LIN {X 0,Y 201.195,Z 1275.243,A -85,B 0,C 180,E1 26164.19,E2 26164.19} C_VEL
LIN {X 0,Y 195.017,Z 1283.497,A -85,B 0,C 180,E1 26183.301,E2 26183.301} C_VEL
LIN {X 0,Y 194.999,Z 1283.507,A -85,B 0,C 180,E1 26196.699,E2 26196.699} C_VEL
LIN {X 0,Y 201.236,Z 1275.253,A -85,B 0,C 180,E1 26215.835,E2 26215.835} C_VEL
LIN {X 0,Y 226.879,Z 1253.045,A -85,B 0,C 180,E1 26235.936,E2 26235.936} C_VEL
LIN {X 0,Y 270.809,Z 1215.708,A -85,B 0,C 180,E1 26251.087,E2 26251.087} C_VEL
LIN {X 0,Y 321.141,Z 1165.252,A -85,B 0,C 180,E1 26260.774,E2 26260.774} C_VEL
LIN {X 0,Y 367.903,Z 1104.901,A -85,B 0,C 180,E1 26266.675,E2 26266.675} C_VEL
LIN {X 0,Y 370.039,Z 1092.442,A -85,B 0,C 180,E1 26272.536,E2 26272.536} C_VEL
LIN {X 0,Y 370.708,Z 1086.535,A -85,B 0,C 180,E1 26278.866,E2 26278.866} C_VEL
LIN {X 0,Y 369.636,Z 1091.478,A -85,B 0,C 180,E1 26286.971,E2 26286.971} C_VEL
LIN {X 0,Y 367.658,Z 1103.886,A -85,B 0,C 180,E1 26293.55,E2 26293.55} C_VEL
LIN {X 0,Y 320.637,Z 1164.15,A -85,B 0,C 180,E1 26299.642,E2 26299.642} C_VEL
LIN {X 0,Y 271.724,Z 1212.598,A -85,B 0,C 180,E1 26309.058,E2 26309.058} C_VEL
LIN {X 0,Y 254.088,Z 1227.944,A -85,B 0,C 180,E1 26313.968,E2 26313.968} C_VEL
LIN {X 0,Y 230.122,Z 1243.335,A -85,B 0,C 180,E1 26319.017,E2 26319.017} C_VEL
LIN {X 0,Y 198.588,Z 1267.683,A -85,B 0,C 180,E1 26338.072,E2 26338.072} C_VEL
LIN {X 0,Y 187.588,Z 1278.356,A -85,B 0,C 180,E1 26358.34,E2 26358.34} C_VEL
LIN {X 0,Y 187.248,Z 1279.786,A -85,B 0,C 180,E1 26372.321,E2 26372.321} C_VEL
LIN {X 0,Y 191.78,Z 1273.585,A -85,B 0,C 180,E1 26393.132,E2 26393.132} C_VEL
LIN {X 0,Y 216.378,Z 1253.744,A -85,B 0,C 180,E1 26414.497,E2 26414.497} C_VEL
LIN {X 0,Y 259.404,Z 1219.732,A -85,B 0,C 180,E1 26430.302,E2 26430.302} C_VEL
LIN {X 0,Y 309.886,Z 1172.58,A -85,B 0,C 180,E1 26440.494,E2 26440.494} C_VEL
LIN {X 0,Y 358.072,Z 1114.769,A -85,B 0,C 180,E1 26446.759,E2 26446.759} C_VEL
LIN {X 0,Y 363.326,Z 1107.025,A -85,B 0,C 180,E1 26447.549,E2 26447.549} C_VEL
LIN {X 0,Y 365.187,Z 1096.26,A -85,B 0,C 180,E1 26454,E2 26454} C_VEL
LIN {X 0,Y 366.009,Z 1093.019,A -85,B 0,C 180,E1 26461.149,E2 26461.149} C_VEL
LIN {X 0,Y 364.774,Z 1102.007,A -85,B 0,C 180,E1 26469.54,E2 26469.54} C_VEL
LIN {X 0,Y 362.75,Z 1109.497,A -85,B 0,C 180,E1 26472.412,E2 26472.412} C_VEL
LIN {X 0,Y 315.401,Z 1168.445,A -85,B 0,C 180,E1 26478.275,E2 26478.275} C_VEL
LIN {X 0,Y 264.142,Z 1217.988,A -85,B 0,C 180,E1 26488.027,E2 26488.027} C_VEL
LIN {X 0,Y 219.314,Z 1254.431,A -85,B 0,C 180,E1 26503.442,E2 26503.442} C_VEL
LIN {X 0,Y 192.773,Z 1276.213,A -85,B 0,C 180,E1 26524.651,E2 26524.651} C_VEL
LIN {X 0,Y 187.008,Z 1283.409,A -85,B 0,C 180,E1 26543.013,E2 26543.013} C_VEL
LIN {X 0,Y 186.992,Z 1283.419,A -85,B 0,C 180,E1 26556.987,E2 26556.987} C_VEL
LIN {X 0,Y 194.576,Z 1274.473,A -85,B 0,C 180,E1 26577.881,E2 26577.881} C_VEL
LIN {X 0,Y 223.086,Z 1251.404,A -85,B 0,C 180,E1 26598.398,E2 26598.398} C_VEL
LIN {X 0,Y 270.344,Z 1212.537,A -85,B 0,C 180,E1 26613.469,E2 26613.469} C_VEL
LIN {X 0,Y 321.331,Z 1162.031,A -85,B 0,C 180,E1 26622.583,E2 26622.583} C_VEL
LIN {X 0,Y 364.275,Z 1106.957,A -85,B 0,C 180,E1 26628.053,E2 26628.053} C_VEL
LIN {X 0,Y 365.739,Z 1094.84,A -85,B 0,C 180,E1 26636.472,E2 26636.472} C_VEL
LIN {X 0,Y 365.521,Z 1094.699,A -85,B 0,C 180,E1 26643.608,E2 26643.608} C_VEL
LIN {X 0,Y 363.417,Z 1106.744,A -85,B 0,C 180,E1 26652.086,E2 26652.086} C_VEL
LIN {X 0,Y 354.781,Z 1119.511,A -85,B 0,C 180,E1 26653.483,E2 26653.483} C_VEL
LIN {X 0,Y 305.533,Z 1177.31,A -85,B 0,C 180,E1 26660.141,E2 26660.141} C_VEL
LIN {X 0,Y 255.501,Z 1223.045,A -85,B 0,C 180,E1 26670.61,E2 26670.61} C_VEL
LIN {X 0,Y 230.122,Z 1243.335,A -85,B 0,C 180,E1 26679.017,E2 26679.017} C_VEL
LIN {X 0,Y 207.484,Z 1256.044,A -85,B 0,C 180,E1 26685.371,E2 26685.371} C_VEL
LIN {X 0,Y 183.024,Z 1274.859,A -85,B 0,C 180,E1 26708.108,E2 26708.108} C_VEL
LIN {X 0,Y 179.002,Z 1279.886,A -85,B 0,C 180,E1 26727.572,E2 26727.572} C_VEL
LIN {X 0,Y 180.111,Z 1277.868,A -85,B 0,C 180,E1 26744.074,E2 26744.074} C_VEL
LIN {X 0,Y 194.472,Z 1265.479,A -85,B 0,C 180,E1 26765.794,E2 26765.794} C_VEL
LIN {X 0,Y 231.406,Z 1238.37,A -85,B 0,C 180,E1 26785.005,E2 26785.005} C_VEL
LIN {X 0,Y 282.219,Z 1196.766,A -85,B 0,C 180,E1 26797.777,E2 26797.777} C_VEL
LIN {X 0,Y 334.047,Z 1143.181,A -85,B 0,C 180,E1 26805.559,E2 26805.559} C_VEL
LIN {X 0,Y 358.451,Z 1111.801,A -85,B 0,C 180,E1 26808.363,E2 26808.363} C_VEL
LIN {X 0,Y 360.648,Z 1100.805,A -85,B 0,C 180,E1 26816.343,E2 26816.343} C_VEL
LIN {X 0,Y 361.231,Z 1099.493,A -85,B 0,C 180,E1 26821.164,E2 26821.164} C_VEL
LIN {X 0,Y 359.753,Z 1108.809,A -85,B 0,C 180,E1 26829.674,E2 26829.674} C_VEL
LIN {X 0,Y 357.604,Z 1114.227,A -85,B 0,C 180,E1 26831.491,E2 26831.491} C_VEL
LIN {X 0,Y 309.713,Z 1171.72,A -85,B 0,C 180,E1 26837.286,E2 26837.286} C_VEL
LIN {X 0,Y 257.526,Z 1220.154,A -85,B 0,C 180,E1 26847.039,E2 26847.039} C_VEL
LIN {X 0,Y 211.366,Z 1255.921,A -85,B 0,C 180,E1 26862.896,E2 26862.896} C_VEL
LIN {X 0,Y 185.522,Z 1275.938,A -85,B 0,C 180,E1 26883.282,E2 26883.282} C_VEL
LIN {X 0,Y 179.001,Z 1283.32,A -85,B 0,C 180,E1 26902.699,E2 26902.699} C_VEL
LIN {X 0,Y 178.986,Z 1283.331,A -85,B 0,C 180,E1 26917.301,E2 26917.301} C_VEL
LIN {X 0,Y 187.317,Z 1274.383,A -85,B 0,C 180,E1 26939.062,E2 26939.062} C_VEL
LIN {X 0,Y 219.732,Z 1249.764,A -85,B 0,C 180,E1 26960.936,E2 26960.936} C_VEL
LIN {X 0,Y 268.261,Z 1211.154,A -85,B 0,C 180,E1 26975.394,E2 26975.394} C_VEL
LIN {X 0,Y 320.449,Z 1160.299,A -85,B 0,C 180,E1 26984.216,E2 26984.216} C_VEL
LIN {X 0,Y 359.366,Z 1111.989,A -85,B 0,C 180,E1 26988.782,E2 26988.782} C_VEL
LIN {X 0,Y 360.904,Z 1101.309,A -85,B 0,C 180,E1 26996.424,E2 26996.424} C_VEL
LIN {X 0,Y 361.206,Z 1099.765,A -85,B 0,C 180,E1 27001.242,E2 27001.242} C_VEL
LIN {X 0,Y 359.072,Z 1109.384,A -85,B 0,C 180,E1 27010.124,E2 27010.124} C_VEL
LIN {X 0,Y 356.374,Z 1114.981,A -85,B 0,C 180,E1 27011.826,E2 27011.826} C_VEL
LIN {X 0,Y 306.687,Z 1173.441,A -85,B 0,C 180,E1 27018.074,E2 27018.074} C_VEL
LIN {X 0,Y 254.942,Z 1220.25,A -85,B 0,C 180,E1 27028.066,E2 27028.066} C_VEL
LIN {X 0,Y 209.353,Z 1254.643,A -85,B 0,C 180,E1 27044.325,E2 27044.325} C_VEL
LIN {X 0,Y 207.484,Z 1256.044,A -85,B 0,C 180,E1 27045.371,E2 27045.371} C_VEL
LIN {X 0,Y 187.092,Z 1266.177,A -85,B 0,C 180,E1 27053.33,E2 27053.33} C_VEL
LIN {X 0,Y 171.751,Z 1278.533,A -85,B 0,C 180,E1 27077.247,E2 27077.247} C_VEL
LIN {X 0,Y 171.202,Z 1279.961,A -85,B 0,C 180,E1 27092.539,E2 27092.539} C_VEL
LIN {X 0,Y 175.429,Z 1274.881,A -85,B 0,C 180,E1 27112.893,E2 27112.893} C_VEL
LIN {X 0,Y 200.894,Z 1256.581,A -85,B 0,C 180,E1 27135.82,E2 27135.82} C_VEL
LIN {X 0,Y 247.578,Z 1223.011,A -85,B 0,C 180,E1 27152.648,E2 27152.648} C_VEL
LIN {X 0,Y 301.387,Z 1176.096,A -85,B 0,C 180,E1 27162.951,E2 27162.951} C_VEL
LIN {X 0,Y 352.482,Z 1117.88,A -85,B 0,C 180,E1 27169.115,E2 27169.115} C_VEL
LIN {X 0,Y 355.572,Z 1108.315,A -85,B 0,C 180,E1 27175.006,E2 27175.006} C_VEL
LIN {X 0,Y 356.408,Z 1105.935,A -85,B 0,C 180,E1 27181.18,E2 27181.18} C_VEL
LIN {X 0,Y 354.546,Z 1115.239,A -85,B 0,C 180,E1 27189.682,E2 27189.682} C_VEL
LIN {X 0,Y 350.481,Z 1121.555,A -85,B 0,C 180,E1 27190.725,E2 27190.725} C_VEL
LIN {X 0,Y 300.864,Z 1178.068,A -85,B 0,C 180,E1 27196.721,E2 27196.721} C_VEL
LIN {X 0,Y 246.815,Z 1225.533,A -85,B 0,C 180,E1 27207.008,E2 27207.008} C_VEL
LIN {X 0,Y 200.187,Z 1259.672,A -85,B 0,C 180,E1 27223.972,E2 27223.972} C_VEL
LIN {X 0,Y 175.136,Z 1278.434,A -85,B 0,C 180,E1 27247.066,E2 27247.066} C_VEL
LIN {X 0,Y 170.978,Z 1283.704,A -85,B 0,C 180,E1 27267.458,E2 27267.458} C_VEL
LIN {X 0,Y 171.647,Z 1282.189,A -85,B 0,C 180,E1 27282.76,E2 27282.76} C_VEL
LIN {X 0,Y 185.284,Z 1270.435,A -85,B 0,C 180,E1 27305.582,E2 27305.582} C_VEL
LIN {X 0,Y 223.656,Z 1243.055,A -85,B 0,C 180,E1 27326.162,E2 27326.162} C_VEL
LIN {X 0,Y 275.987,Z 1201.491,A -85,B 0,C 180,E1 27339.198,E2 27339.198} C_VEL
LIN {X 0,Y 328.939,Z 1148.262,A -85,B 0,C 180,E1 27346.968,E2 27346.968} C_VEL
LIN {X 0,Y 354.471,Z 1116.219,A -85,B 0,C 180,E1 27349.881,E2 27349.881} C_VEL
LIN {X 0,Y 356.56,Z 1106.115,A -85,B 0,C 180,E1 27358.821,E2 27358.821} C_VEL
LIN {X 0,Y 354.841,Z 1111.535,A -85,B 0,C 180,E1 27367.41,E2 27367.41} C_VEL
LIN {X 0,Y 352.623,Z 1117.947,A -85,B 0,C 180,E1 27370.75,E2 27370.75} C_VEL
LIN {X 0,Y 301.319,Z 1176.4,A -85,B 0,C 180,E1 27377.008,E2 27377.008} C_VEL
LIN {X 0,Y 247.419,Z 1223.224,A -85,B 0,C 180,E1 27387.282,E2 27387.282} C_VEL
LIN {X 0,Y 200.777,Z 1256.725,A -85,B 0,C 180,E1 27404.146,E2 27404.146} C_VEL
LIN {X 0,Y 187.092,Z 1266.177,A -85,B 0,C 180,E1 27413.33,E2 27413.33} C_VEL
LIN {X 0,Y 169.798,Z 1273.66,A -85,B 0,C 180,E1 27423.03,E2 27423.03} C_VEL
LIN {X 0,Y 163.094,Z 1279.631,A -85,B 0,C 180,E1 27441.983,E2 27441.983} C_VEL
LIN {X 0,Y 163.159,Z 1279.601,A -85,B 0,C 180,E1 27458.015,E2 27458.015} C_VEL
LIN {X 0,Y 173.522,Z 1270.917,A -85,B 0,C 180,E1 27481.627,E2 27481.627} C_VEL
LIN {X 0,Y 210.173,Z 1246.793,A -85,B 0,C 180,E1 27504.269,E2 27504.269} C_VEL
LIN {X 0,Y 262.077,Z 1208.946,A -85,B 0,C 180,E1 27518.303,E2 27518.303} C_VEL
LIN {X 0,Y 316.745,Z 1158.307,A -85,B 0,C 180,E1 27526.782,E2 27526.782} C_VEL
LIN {X 0,Y 348.764,Z 1120.766,A -85,B 0,C 180,E1 27530.367,E2 27530.367} C_VEL
LIN {X 0,Y 351.543,Z 1112.083,A -85,B 0,C 180,E1 27538.724,E2 27538.724} C_VEL
LIN {X 0,Y 350.398,Z 1116.362,A -85,B 0,C 180,E1 27546.173,E2 27546.173} C_VEL
LIN {X 0,Y 348.485,Z 1122.201,A -85,B 0,C 180,E1 27549.453,E2 27549.453} C_VEL
LIN {X 0,Y 296.939,Z 1179.584,A -85,B 0,C 180,E1 27555.422,E2 27555.422} C_VEL
LIN {X 0,Y 241.164,Z 1226.947,A -85,B 0,C 180,E1 27565.712,E2 27565.712} C_VEL
LIN {X 0,Y 194.488,Z 1259.579,A -85,B 0,C 180,E1 27582.202,E2 27582.202} C_VEL
LIN {X 0,Y 167.582,Z 1278.344,A -85,B 0,C 180,E1 27605.969,E2 27605.969} C_VEL
LIN {X 0,Y 162.958,Z 1283.617,A -85,B 0,C 180,E1 27627.333,E2 27627.333} C_VEL
LIN {X 0,Y 163.819,Z 1282.005,A -85,B 0,C 180,E1 27643.871,E2 27643.871} C_VEL
LIN {X 0,Y 180.769,Z 1268.817,A -85,B 0,C 180,E1 27668.991,E2 27668.991} C_VEL
LIN {X 0,Y 221.546,Z 1241.207,A -85,B 0,C 180,E1 27688.832,E2 27688.832} C_VEL
LIN {X 0,Y 275.798,Z 1199.137,A -85,B 0,C 180,E1 27701.284,E2 27701.284} C_VEL
LIN {X 0,Y 329.387,Z 1145.675,A -85,B 0,C 180,E1 27708.631,E2 27708.631} C_VEL
LIN {X 0,Y 349.546,Z 1120.838,A -85,B 0,C 180,E1 27710.854,E2 27710.854} C_VEL
LIN {X 0,Y 351.639,Z 1112.474,A -85,B 0,C 180,E1 27718.804,E2 27718.804} C_VEL
LIN {X 0,Y 350.023,Z 1116.409,A -85,B 0,C 180,E1 27726.261,E2 27726.261} C_VEL
LIN {X 0,Y 347.621,Z 1122.721,A -85,B 0,C 180,E1 27729.781,E2 27729.781} C_VEL
LIN {X 0,Y 295.744,Z 1179.677,A -85,B 0,C 180,E1 27735.956,E2 27735.956} C_VEL
LIN {X 0,Y 241.553,Z 1224.963,A -85,B 0,C 180,E1 27746.058,E2 27746.058} C_VEL
LIN {X 0,Y 193.133,Z 1258.137,A -85,B 0,C 180,E1 27763.42,E2 27763.42} C_VEL
LIN {X 0,Y 169.798,Z 1273.66,A -85,B 0,C 180,E1 27783.03,E2 27783.03} C_VEL
LIN {X 0,Y 156.267,Z 1278.321,A -85,B 0,C 180,E1 27794.526,E2 27794.526} C_VEL
LIN {X 0,Y 155.168,Z 1280.137,A -85,B 0,C 180,E1 27812.801,E2 27812.801} C_VEL
LIN {X 0,Y 161.274,Z 1274.488,A -85,B 0,C 180,E1 27836.473,E2 27836.473} C_VEL
LIN {X 0,Y 194.237,Z 1253.968,A -85,B 0,C 180,E1 27861.528,E2 27861.528} C_VEL
LIN {X 0,Y 244.846,Z 1219.958,A -85,B 0,C 180,E1 27877.122,E2 27877.122} C_VEL
LIN {X 0,Y 300.305,Z 1173.094,A -85,B 0,C 180,E1 27886.44,E2 27886.44} C_VEL
LIN {X 0,Y 343.984,Z 1125.372,A -85,B 0,C 180,E1 27891.399,E2 27891.399} C_VEL
LIN {X 0,Y 346.418,Z 1118.322,A -85,B 0,C 180,E1 27898.705,E2 27898.705} C_VEL
LIN {X 0,Y 345.169,Z 1122.764,A -85,B 0,C 180,E1 27906.267,E2 27906.267} C_VEL
LIN {X 0,Y 343.768,Z 1126.608,A -85,B 0,C 180,E1 27908.435,E2 27908.435} C_VEL
LIN {X 0,Y 291.229,Z 1182.986,A -85,B 0,C 180,E1 27914.361,E2 27914.361} C_VEL
LIN {X 0,Y 235.946,Z 1228.133,A -85,B 0,C 180,E1 27924.283,E2 27924.283} C_VEL
LIN {X 0,Y 186.895,Z 1260.839,A -85,B 0,C 180,E1 27941.359,E2 27941.359} C_VEL
LIN {X 0,Y 160.09,Z 1278.253,A -85,B 0,C 180,E1 27964.768,E2 27964.768} C_VEL
LIN {X 0,Y 154.936,Z 1283.529,A -85,B 0,C 180,E1 27987.195,E2 27987.195} C_VEL
LIN {X 0,Y 155.862,Z 1282.011,A -85,B 0,C 180,E1 28004.078,E2 28004.078} C_VEL
LIN {X 0,Y 172.151,Z 1270.141,A -85,B 0,C 180,E1 28028.962,E2 28028.962} C_VEL
LIN {X 0,Y 214.695,Z 1242.871,A -85,B 0,C 180,E1 28049.916,E2 28049.916} C_VEL
LIN {X 0,Y 270.961,Z 1200.936,A -85,B 0,C 180,E1 28062.579,E2 28062.579} C_VEL
LIN {X 0,Y 326.907,Z 1146.64,A -85,B 0,C 180,E1 28069.95,E2 28069.95} C_VEL
LIN {X 0,Y 344.662,Z 1125.488,A -85,B 0,C 180,E1 28071.896,E2 28071.896} C_VEL
LIN {X 0,Y 346.513,Z 1118.711,A -85,B 0,C 180,E1 28078.786,E2 28078.786} C_VEL
LIN {X 0,Y 344.788,Z 1122.817,A -85,B 0,C 180,E1 28086.356,E2 28086.356} C_VEL
LIN {X 0,Y 342.867,Z 1127.123,A -85,B 0,C 180,E1 28088.759,E2 28088.759} C_VEL
LIN {X 0,Y 289.1,Z 1183.852,A -85,B 0,C 180,E1 28095.015,E2 28095.015} C_VEL
LIN {X 0,Y 232.169,Z 1229.12,A -85,B 0,C 180,E1 28105.638,E2 28105.638} C_VEL
LIN {X 0,Y 183.612,Z 1260.51,A -85,B 0,C 180,E1 28123.722,E2 28123.722} C_VEL
LIN {X 0,Y 158.982,Z 1276.302,A -85,B 0,C 180,E1 28147.57,E2 28147.57} C_VEL
LIN {X 0,Y 156.267,Z 1278.321,A -85,B 0,C 180,E1 28154.526,E2 28154.526} C_VEL
LIN {X 0,Y 146.914,Z 1280.235,A -85,B 0,C 180,E1 28167.516,E2 28167.516} C_VEL
LIN {X 0,Y 148.18,Z 1278.77,A -85,B 0,C 180,E1 28184.825,E2 28184.825} C_VEL
LIN {X 0,Y 165.314,Z 1267.75,A -85,B 0,C 180,E1 28209.953,E2 28209.953} C_VEL
LIN {X 0,Y 208.556,Z 1242.191,A -85,B 0,C 180,E1 28230.761,E2 28230.761} C_VEL
LIN {X 0,Y 265.721,Z 1201.741,A -85,B 0,C 180,E1 28243.402,E2 28243.402} C_VEL
LIN {X 0,Y 321.32,Z 1150.153,A -85,B 0,C 180,E1 28250.545,E2 28250.545} C_VEL
LIN {X 0,Y 339.042,Z 1129.89,A -85,B 0,C 180,E1 28252.482,E2 28252.482} C_VEL
LIN {X 0,Y 341.255,Z 1124.682,A -85,B 0,C 180,E1 28260.805,E2 28260.805} C_VEL
LIN {X 0,Y 338.694,Z 1131.184,A -85,B 0,C 180,E1 28267.412,E2 28267.412} C_VEL
LIN {X 0,Y 284.233,Z 1187.296,A -85,B 0,C 180,E1 28273.42,E2 28273.42} C_VEL
LIN {X 0,Y 227.106,Z 1231.739,A -85,B 0,C 180,E1 28283.658,E2 28283.658} C_VEL
LIN {X 0,Y 177.311,Z 1263.096,A -85,B 0,C 180,E1 28301.549,E2 28301.549} C_VEL
LIN {X 0,Y 151.147,Z 1279.385,A -85,B 0,C 180,E1 28326.338,E2 28326.338} C_VEL
LIN {X 0,Y 146.914,Z 1283.441,A -85,B 0,C 180,E1 28347.041,E2 28347.041} C_VEL
LIN {X 0,Y 147.995,Z 1281.923,A -85,B 0,C 180,E1 28364.843,E2 28364.843} C_VEL
LIN {X 0,Y 168.083,Z 1268.635,A -85,B 0,C 180,E1 28392.585,E2 28392.585} C_VEL
LIN {X 0,Y 213.321,Z 1241.025,A -85,B 0,C 180,E1 28412.703,E2 28412.703} C_VEL
LIN {X 0,Y 271.233,Z 1198.685,A -85,B 0,C 180,E1 28424.686,E2 28424.686} C_VEL
LIN {X 0,Y 327.503,Z 1144.437,A -85,B 0,C 180,E1 28431.575,E2 28431.575} C_VEL
LIN {X 0,Y 339.627,Z 1130.078,A -85,B 0,C 180,E1 28432.994,E2 28432.994} C_VEL
LIN {X 0,Y 341.24,Z 1124.941,A -85,B 0,C 180,E1 28440.615,E2 28440.615} C_VEL
LIN {X 0,Y 338.878,Z 1130.436,A -85,B 0,C 180,E1 28447.529,E2 28447.529} C_VEL
LIN {X 0,Y 284.419,Z 1186.22,A -85,B 0,C 180,E1 28453.76,E2 28453.76} C_VEL
LIN {X 0,Y 226.913,Z 1230.379,A -85,B 0,C 180,E1 28464.17,E2 28464.17} C_VEL
LIN {X 0,Y 175.98,Z 1261.736,A -85,B 0,C 180,E1 28482.904,E2 28482.904} C_VEL
LIN {X 0,Y 150.076,Z 1277.237,A -85,B 0,C 180,E1 28509.288,E2 28509.288} C_VEL
LIN {X 0,Y 146.914,Z 1280.235,A -85,B 0,C 180,E1 28527.516,E2 28527.516} C_VEL
LIN {X 0,Y 139.41,Z 1279.532,A -85,B 0,C 180,E1 28541.496,E2 28541.496} C_VEL
LIN {X 0,Y 155.826,Z 1269.649,A -85,B 0,C 180,E1 28569.242,E2 28569.242} C_VEL
LIN {X 0,Y 199.179,Z 1245.552,A -85,B 0,C 180,E1 28591.117,E2 28591.117} C_VEL
LIN {X 0,Y 257.986,Z 1206.184,A -85,B 0,C 180,E1 28604.278,E2 28604.278} C_VEL
LIN {X 0,Y 316.518,Z 1154.072,A -85,B 0,C 180,E1 28611.654,E2 28611.654} C_VEL
LIN {X 0,Y 334.007,Z 1134.744,A -85,B 0,C 180,E1 28613.438,E2 28613.438} C_VEL
LIN {X 0,Y 335.952,Z 1130.602,A -85,B 0,C 180,E1 28618.664,E2 28618.664} C_VEL
LIN {X 0,Y 334.42,Z 1134.828,A -85,B 0,C 180,E1 28626.142,E2 28626.142} C_VEL
LIN {X 0,Y 277.384,Z 1191.533,A -85,B 0,C 180,E1 28632.432,E2 28632.432} C_VEL
LIN {X 0,Y 218.28,Z 1235.316,A -85,B 0,C 180,E1 28642.991,E2 28642.991} C_VEL
LIN {X 0,Y 169.75,Z 1264.166,A -85,B 0,C 180,E1 28660.59,E2 28660.59} C_VEL
LIN {X 0,Y 142.215,Z 1280.182,A -85,B 0,C 180,E1 28688.085,E2 28688.085} C_VEL
LIN {X 0,Y 138.905,Z 1283.353,A -85,B 0,C 180,E1 28706.87,E2 28706.87} C_VEL
LIN {X 0,Y 140.139,Z 1281.834,A -85,B 0,C 180,E1 28725.696,E2 28725.696} C_VEL
LIN {X 0,Y 158.595,Z 1270.499,A -85,B 0,C 180,E1 28752.017,E2 28752.017} C_VEL
LIN {X 0,Y 205.375,Z 1243.558,A -85,B 0,C 180,E1 28773.563,E2 28773.563} C_VEL
LIN {X 0,Y 264.133,Z 1202.601,A -85,B 0,C 180,E1 28785.67,E2 28785.67} C_VEL
LIN {X 0,Y 321.204,Z 1149.944,A -85,B 0,C 180,E1 28792.521,E2 28792.521} C_VEL
LIN {X 0,Y 334.47,Z 1135.059,A -85,B 0,C 180,E1 28793.858,E2 28793.858} C_VEL
LIN {X 0,Y 335.817,Z 1131.076,A -85,B 0,C 180,E1 28801.336,E2 28801.336} C_VEL
LIN {X 0,Y 332.534,Z 1136.844,A -85,B 0,C 180,E1 28806.743,E2 28806.743} C_VEL
LIN {X 0,Y 276.142,Z 1191.82,A -85,B 0,C 180,E1 28813,E2 28813} C_VEL
LIN {X 0,Y 218.878,Z 1233.575,A -85,B 0,C 180,E1 28823.358,E2 28823.358} C_VEL
LIN {X 0,Y 168.05,Z 1263.152,A -85,B 0,C 180,E1 28842.206,E2 28842.206} C_VEL
LIN {X 0,Y 142.461,Z 1277.326,A -85,B 0,C 180,E1 28868.125,E2 28868.125} C_VEL
LIN {X 0,Y 138.887,Z 1280.323,A -85,B 0,C 180,E1 28887.418,E2 28887.418} C_VEL
LIN {X 0,Y 139.41,Z 1279.532,A -85,B 0,C 180,E1 28901.496,E2 28901.496} C_VEL
LIN {X 0,Y 136.452,Z 1276.545,A -85,B 0,C 180,E1 28916.168,E2 28916.168} C_VEL
LIN {X 0,Y 171.443,Z 1258.694,A -85,B 0,C 180,E1 28944.33,E2 28944.33} C_VEL
LIN {X 0,Y 227.496,Z 1226.156,A -85,B 0,C 180,E1 28961.07,E2 28961.07} C_VEL
LIN {X 0,Y 287.562,Z 1180.546,A -85,B 0,C 180,E1 28970.248,E2 28970.248} C_VEL
LIN {X 0,Y 329.132,Z 1139.395,A -85,B 0,C 180,E1 28974.666,E2 28974.666} C_VEL
LIN {X 0,Y 330.526,Z 1136.788,A -85,B 0,C 180,E1 28981.272,E2 28981.272} C_VEL
LIN {X 0,Y 328.525,Z 1140.754,A -85,B 0,C 180,E1 28985.322,E2 28985.322} C_VEL
LIN {X 0,Y 270.712,Z 1195.661,A -85,B 0,C 180,E1 28991.375,E2 28991.375} C_VEL
LIN {X 0,Y 209.11,Z 1238.993,A -85,B 0,C 180,E1 29002.38,E2 29002.38} C_VEL
LIN {X 0,Y 159.07,Z 1266.951,A -85,B 0,C 180,E1 29021.377,E2 29021.377} C_VEL
LIN {X 0,Y 134.657,Z 1280.092,A -85,B 0,C 180,E1 29046.785,E2 29046.785} C_VEL
LIN {X 0,Y 130.881,Z 1283.265,A -85,B 0,C 180,E1 29066.678,E2 29066.678} C_VEL
LIN {X 0,Y 132.327,Z 1281.745,A -85,B 0,C 180,E1 29086.649,E2 29086.649} C_VEL
LIN {X 0,Y 152.475,Z 1270.408,A -85,B 0,C 180,E1 29114.125,E2 29114.125} C_VEL
LIN {X 0,Y 201.405,Z 1243.688,A -85,B 0,C 180,E1 29135.603,E2 29135.603} C_VEL
LIN {X 0,Y 262.201,Z 1202.513,A -85,B 0,C 180,E1 29147.429,E2 29147.429} C_VEL
LIN {X 0,Y 320.231,Z 1149.856,A -85,B 0,C 180,E1 29153.992,E2 29153.992} C_VEL
LIN {X 0,Y 329.451,Z 1139.81,A -85,B 0,C 180,E1 29155.011,E2 29155.011} C_VEL
LIN {X 0,Y 330.414,Z 1137.075,A -85,B 0,C 180,E1 29161.358,E2 29161.358} C_VEL
LIN {X 0,Y 327.668,Z 1141.474,A -85,B 0,C 180,E1 29165.688,E2 29165.688} C_VEL
LIN {X 0,Y 269.343,Z 1195.997,A -85,B 0,C 180,E1 29171.959,E2 29171.959} C_VEL
LIN {X 0,Y 209.726,Z 1237.359,A -85,B 0,C 180,E1 29182.787,E2 29182.787} C_VEL
LIN {X 0,Y 160.681,Z 1264.266,A -85,B 0,C 180,E1 29201.115,E2 29201.115} C_VEL
LIN {X 0,Y 134.903,Z 1277.416,A -85,B 0,C 180,E1 29226.83,E2 29226.83} C_VEL
LIN {X 0,Y 130.914,Z 1280.412,A -85,B 0,C 180,E1 29246.68,E2 29246.68} C_VEL
LIN {X 0,Y 132.527,Z 1278.948,A -85,B 0,C 180,E1 29266.624,E2 29266.624} C_VEL
LIN {X 0,Y 136.452,Z 1276.545,A -85,B 0,C 180,E1 29276.168,E2 29276.168} C_VEL
LIN {X 0,Y 140.06,Z 1271.301,A -85,B 0,C 180,E1 29290.712,E2 29290.712} C_VEL
LIN {X 0,Y 186.683,Z 1248.373,A -85,B 0,C 180,E1 29314.029,E2 29314.029} C_VEL
LIN {X 0,Y 247.881,Z 1210.661,A -85,B 0,C 180,E1 29327.007,E2 29327.007} C_VEL
LIN {X 0,Y 308.358,Z 1160.282,A -85,B 0,C 180,E1 29334.086,E2 29334.086} C_VEL
LIN {X 0,Y 323.904,Z 1144.401,A -85,B 0,C 180,E1 29335.583,E2 29335.583} C_VEL
LIN {X 0,Y 325.054,Z 1142.71,A -85,B 0,C 180,E1 29341.294,E2 29341.294} C_VEL
LIN {X 0,Y 322.953,Z 1145.849,A -85,B 0,C 180,E1 29344.261,E2 29344.261} C_VEL
LIN {X 0,Y 263.951,Z 1199.577,A -85,B 0,C 180,E1 29350.287,E2 29350.287} C_VEL
LIN {X 0,Y 202.984,Z 1240.653,A -85,B 0,C 180,E1 29360.948,E2 29360.948} C_VEL
LIN {X 0,Y 150.53,Z 1268.309,A -85,B 0,C 180,E1 29380.922,E2 29380.922} C_VEL
LIN {X 0,Y 127.143,Z 1280.002,A -85,B 0,C 180,E1 29405.324,E2 29405.324} C_VEL
LIN {X 0,Y 122.857,Z 1283.177,A -85,B 0,C 180,E1 29426.461,E2 29426.461} C_VEL
LIN {X 0,Y 124.538,Z 1281.656,A -85,B 0,C 180,E1 29447.724,E2 29447.724} C_VEL
LIN {X 0,Y 146.586,Z 1270.318,A -85,B 0,C 180,E1 29476.402,E2 29476.402} C_VEL
LIN {X 0,Y 198.08,Z 1243.597,A -85,B 0,C 180,E1 29497.819,E2 29497.819} C_VEL
LIN {X 0,Y 260.501,Z 1202.423,A -85,B 0,C 180,E1 29509.233,E2 29509.233} C_VEL
LIN {X 0,Y 319.934,Z 1149.281,A -85,B 0,C 180,E1 29515.509,E2 29515.509} C_VEL
LIN {X 0,Y 324.216,Z 1144.711,A -85,B 0,C 180,E1 29516.019,E2 29516.019} C_VEL
LIN {X 0,Y 324.903,Z 1142.997,A -85,B 0,C 180,E1 29521.381,E2 29521.381} C_VEL
LIN {X 0,Y 322.828,Z 1145.866,A -85,B 0,C 180,E1 29524.596,E2 29524.596} C_VEL
LIN {X 0,Y 264.259,Z 1198.727,A -85,B 0,C 180,E1 29530.651,E2 29530.651} C_VEL
LIN {X 0,Y 203.563,Z 1239.174,A -85,B 0,C 180,E1 29541.371,E2 29541.371} C_VEL
LIN {X 0,Y 151.179,Z 1266.214,A -85,B 0,C 180,E1 29561.206,E2 29561.206} C_VEL
LIN {X 0,Y 124.682,Z 1279.065,A -85,B 0,C 180,E1 29592.297,E2 29592.297} C_VEL
LIN {X 0,Y 123.097,Z 1280.489,A -85,B 0,C 180,E1 29613.532,E2 29613.532} C_VEL
LIN {X 0,Y 133.983,Z 1274.233,A -85,B 0,C 180,E1 29644.468,E2 29644.468} C_VEL
LIN {X 0,Y 140.06,Z 1271.301,A -85,B 0,C 180,E1 29650.712,E2 29650.712} C_VEL
LIN {X 0,Y 150.441,Z 1264.214,A -85,B 0,C 180,E1 29663.852,E2 29663.852} C_VEL
LIN {X 0,Y 207.041,Z 1235.613,A -85,B 0,C 180,E1 29682.219,E2 29682.219} C_VEL
LIN {X 0,Y 269.348,Z 1193.708,A -85,B 0,C 180,E1 29691.853,E2 29691.853} C_VEL
LIN {X 0,Y 318.654,Z 1149.326,A -85,B 0,C 180,E1 29696.823,E2 29696.823} C_VEL
LIN {X 0,Y 318.824,Z 1149.441,A -85,B 0,C 180,E1 29702.859,E2 29702.859} C_VEL
LIN {X 0,Y 258.114,Z 1202.872,A -85,B 0,C 180,E1 29709.052,E2 29709.052} C_VEL
LIN {X 0,Y 195.289,Z 1243.278,A -85,B 0,C 180,E1 29719.846,E2 29719.846} C_VEL
LIN {X 0,Y 140.875,Z 1270.198,A -85,B 0,C 180,E1 29741.161,E2 29741.161} C_VEL
LIN {X 0,Y 116.789,Z 1281.552,A -85,B 0,C 180,E1 29771.056,E2 29771.056} C_VEL
LIN {X 0,Y 114.787,Z 1283.093,A -85,B 0,C 180,E1 29793.787,E2 29793.787} C_VEL
LIN {X 0,Y 124.074,Z 1277.834,A -85,B 0,C 180,E1 29823.368,E2 29823.368} C_VEL
LIN {X 0,Y 167.664,Z 1257.751,A -85,B 0,C 180,E1 29851.872,E2 29851.872} C_VEL
LIN {X 0,Y 229.532,Z 1222.906,A -85,B 0,C 180,E1 29866.885,E2 29866.885} C_VEL
LIN {X 0,Y 291.777,Z 1175.648,A -85,B 0,C 180,E1 29874.599,E2 29874.599} C_VEL
LIN {X 0,Y 318.848,Z 1149.706,A -85,B 0,C 180,E1 29877.097,E2 29877.097} C_VEL
LIN {X 0,Y 318.096,Z 1150.27,A -85,B 0,C 180,E1 29883.461,E2 29883.461} C_VEL
LIN {X 0,Y 257.568,Z 1202.777,A -85,B 0,C 180,E1 29889.522,E2 29889.522} C_VEL
LIN {X 0,Y 194.372,Z 1242.755,A -85,B 0,C 180,E1 29900.639,E2 29900.639} C_VEL
LIN {X 0,Y 141.514,Z 1268.207,A -85,B 0,C 180,E1 29921.396,E2 29921.396} C_VEL
LIN {X 0,Y 116.96,Z 1279.154,A -85,B 0,C 180,E1 29951.086,E2 29951.086} C_VEL
LIN {X 0,Y 115.068,Z 1280.577,A -85,B 0,C 180,E1 29973.779,E2 29973.779} C_VEL
LIN {X 0,Y 127.271,Z 1274.324,A -85,B 0,C 180,E1 30006.569,E2 30006.569} C_VEL
LIN {X 0,Y 150.441,Z 1264.214,A -85,B 0,C 180,E1 30023.852,E2 30023.852} C_VEL
LIN {X 0,Y 166.641,Z 1254.962,A -85,B 0,C 180,E1 30034.835,E2 30034.835} C_VEL
LIN {X 0,Y 229.885,Z 1220.605,A -85,B 0,C 180,E1 30048.708,E2 30048.708} C_VEL
LIN {X 0,Y 292.205,Z 1174.056,A -85,B 0,C 180,E1 30055.897,E2 30055.897} C_VEL
LIN {X 0,Y 313.363,Z 1154.488,A -85,B 0,C 180,E1 30057.813,E2 30057.813} C_VEL
LIN {X 0,Y 312.34,Z 1155.735,A -85,B 0,C 180,E1 30062.027,E2 30062.027} C_VEL
LIN {X 0,Y 249.881,Z 1207.946,A -85,B 0,C 180,E1 30068.067,E2 30068.067} C_VEL
LIN {X 0,Y 184.826,Z 1247.299,A -85,B 0,C 180,E1 30079.334,E2 30079.334} C_VEL
LIN {X 0,Y 131.29,Z 1271.935,A -85,B 0,C 180,E1 30101.338,E2 30101.338} C_VEL
LIN {X 0,Y 109.094,Z 1281.463,A -85,B 0,C 180,E1 30129.663,E2 30129.663} C_VEL
LIN {X 0,Y 106.782,Z 1283.005,A -85,B 0,C 180,E1 30154.072,E2 30154.072} C_VEL
LIN {X 0,Y 117.26,Z 1277.744,A -85,B 0,C 180,E1 30185.59,E2 30185.59} C_VEL
LIN {X 0,Y 163.245,Z 1257.96,A -85,B 0,C 180,E1 30214.24,E2 30214.24} C_VEL
LIN {X 0,Y 225.726,Z 1224.116,A -85,B 0,C 180,E1 30228.625,E2 30228.625} C_VEL
LIN {X 0,Y 290.126,Z 1176.42,A -85,B 0,C 180,E1 30236.139,E2 30236.139} C_VEL
LIN {X 0,Y 313.649,Z 1154.622,A -85,B 0,C 180,E1 30238.33,E2 30238.33} C_VEL
LIN {X 0,Y 312.245,Z 1155.898,A -85,B 0,C 180,E1 30242.388,E2 30242.388} C_VEL
LIN {X 0,Y 250.619,Z 1207.002,A -85,B 0,C 180,E1 30248.379,E2 30248.379} C_VEL
LIN {X 0,Y 188.455,Z 1244.543,A -85,B 0,C 180,E1 30259.037,E2 30259.037} C_VEL
LIN {X 0,Y 131.798,Z 1270.088,A -85,B 0,C 180,E1 30281.59,E2 30281.59} C_VEL
LIN {X 0,Y 109.282,Z 1279.243,A -85,B 0,C 180,E1 30309.701,E2 30309.701} C_VEL
LIN {X 0,Y 107.044,Z 1280.665,A -85,B 0,C 180,E1 30334.062,E2 30334.062} C_VEL
LIN {X 0,Y 120.723,Z 1274.415,A -85,B 0,C 180,E1 30368.911,E2 30368.911} C_VEL
LIN {X 0,Y 166.641,Z 1254.962,A -85,B 0,C 180,E1 30394.835,E2 30394.835} C_VEL
LIN {X 0,Y 186.864,Z 1243.975,A -85,B 0,C 180,E1 30403.62,E2 30403.62} C_VEL
LIN {X 0,Y 253.228,Z 1204.296,A -85,B 0,C 180,E1 30413.882,E2 30413.882} C_VEL
LIN {X 0,Y 307.875,Z 1159.554,A -85,B 0,C 180,E1 30418.895,E2 30418.895} C_VEL
LIN {X 0,Y 306.784,Z 1160.665,A -85,B 0,C 180,E1 30420.88,E2 30420.88} C_VEL
LIN {X 0,Y 244.3,Z 1210.897,A -85,B 0,C 180,E1 30426.672,E2 30426.672} C_VEL
LIN {X 0,Y 178.894,Z 1248.806,A -85,B 0,C 180,E1 30437.632,E2 30437.632} C_VEL
LIN {X 0,Y 121.64,Z 1273.435,A -85,B 0,C 180,E1 30461.578,E2 30461.578} C_VEL
LIN {X 0,Y 99.398,Z 1282.434,A -85,B 0,C 180,E1 30496.77,E2 30496.77} C_VEL
LIN {X 0,Y 99.4,Z 1282.449,A -85,B 0,C 180,E1 30523.229,E2 30523.229} C_VEL
LIN {X 0,Y 121.643,Z 1273.482,A -85,B 0,C 180,E1 30558.419,E2 30558.419} C_VEL
LIN {X 0,Y 178.921,Z 1248.894,A -85,B 0,C 180,E1 30582.366,E2 30582.366} C_VEL
LIN {X 0,Y 244.227,Z 1211.109,A -85,B 0,C 180,E1 30593.319,E2 30593.319} C_VEL
LIN {X 0,Y 306.793,Z 1160.918,A -85,B 0,C 180,E1 30599.104,E2 30599.104} C_VEL
LIN {X 0,Y 306.565,Z 1161.042,A -85,B 0,C 180,E1 30601.268,E2 30601.268} C_VEL
LIN {X 0,Y 243.812,Z 1210.891,A -85,B 0,C 180,E1 30607.138,E2 30607.138} C_VEL
LIN {X 0,Y 179.473,Z 1247.67,A -85,B 0,C 180,E1 30618.082,E2 30618.082} C_VEL
LIN {X 0,Y 122.067,Z 1271.721,A -85,B 0,C 180,E1 30641.805,E2 30641.805} C_VEL
LIN {X 0,Y 99.526,Z 1280.336,A -85,B 0,C 180,E1 30676.788,E2 30676.788} C_VEL
LIN {X 0,Y 99.593,Z 1280.31,A -85,B 0,C 180,E1 30703.204,E2 30703.204} C_VEL
LIN {X 0,Y 122.055,Z 1271.649,A -85,B 0,C 180,E1 30738.203,E2 30738.203} C_VEL
LIN {X 0,Y 176.267,Z 1249.058,A -85,B 0,C 180,E1 30761.157,E2 30761.157} C_VEL
LIN {X 0,Y 186.864,Z 1243.975,A -85,B 0,C 180,E1 30763.62,E2 30763.62} C_VEL
LIN {X 0,Y 209.945,Z 1230.845,A -85,B 0,C 180,E1 30770.439,E2 30770.439} C_VEL
LIN {X 0,Y 276.937,Z 1186.217,A -85,B 0,C 180,E1 30778.004,E2 30778.004} C_VEL
LIN {X 0,Y 300.269,Z 1166.599,A -85,B 0,C 180,E1 30779.783,E2 30779.783} C_VEL
LIN {X 0,Y 236.168,Z 1215.649,A -85,B 0,C 180,E1 30785.542,E2 30785.542} C_VEL
LIN {X 0,Y 169.824,Z 1251.883,A -85,B 0,C 180,E1 30796.615,E2 30796.615} C_VEL
LIN {X 0,Y 111.919,Z 1274.934,A -85,B 0,C 180,E1 30821.817,E2 30821.817} C_VEL
LIN {X 0,Y 91.513,Z 1282.345,A -85,B 0,C 180,E1 30855.606,E2 30855.606} C_VEL
LIN {X 0,Y 91.516,Z 1282.361,A -85,B 0,C 180,E1 30884.392,E2 30884.392} C_VEL
LIN {X 0,Y 116.254,Z 1273.391,A -85,B 0,C 180,E1 30921.508,E2 30921.508} C_VEL
LIN {X 0,Y 176.389,Z 1248.88,A -85,B 0,C 180,E1 30944.933,E2 30944.933} C_VEL
LIN {X 0,Y 244.758,Z 1210.124,A -85,B 0,C 180,E1 30955.406,E2 30955.406} C_VEL
LIN {X 0,Y 298.469,Z 1168.527,A -85,B 0,C 180,E1 30960.286,E2 30960.286} C_VEL
LIN {X 0,Y 232.707,Z 1217.642,A -85,B 0,C 180,E1 30966.368,E2 30966.368} C_VEL
LIN {X 0,Y 167.251,Z 1252.319,A -85,B 0,C 180,E1 30977.81,E2 30977.81} C_VEL
LIN {X 0,Y 112.313,Z 1273.355,A -85,B 0,C 180,E1 31002.043,E2 31002.043} C_VEL
LIN {X 0,Y 91.65,Z 1280.424,A -85,B 0,C 180,E1 31035.629,E2 31035.629} C_VEL
LIN {X 0,Y 91.717,Z 1280.399,A -85,B 0,C 180,E1 31064.361,E2 31064.361} C_VEL
LIN {X 0,Y 116.681,Z 1271.74,A -85,B 0,C 180,E1 31101.246,E2 31101.246} C_VEL
LIN {X 0,Y 173.745,Z 1249.151,A -85,B 0,C 180,E1 31123.769,E2 31123.769} C_VEL
LIN {X 0,Y 209.945,Z 1230.845,A -85,B 0,C 180,E1 31130.439,E2 31130.439} C_VEL
LIN {X 0,Y 234.416,Z 1216,A -85,B 0,C 180,E1 31135.892,E2 31135.892} C_VEL
LIN {X 0,Y 277.406,Z 1185.824,A -85,B 0,C 180,E1 31139.78,E2 31139.78} C_VEL
LIN {X 0,Y 210.029,Z 1230.654,A -85,B 0,C 180,E1 31146.522,E2 31146.522} C_VEL
LIN {X 0,Y 142.031,Z 1262.355,A -85,B 0,C 180,E1 31160.887,E2 31160.887} C_VEL
LIN {X 0,Y 94.511,Z 1278.66,A -85,B 0,C 180,E1 31190.07,E2 31190.07} C_VEL
LIN {X 0,Y 82.811,Z 1282.737,A -85,B 0,C 180,E1 31224.746,E2 31224.746} C_VEL
LIN {X 0,Y 86.55,Z 1281.211,A -85,B 0,C 180,E1 31255.979,E2 31255.979} C_VEL
LIN {X 0,Y 123.674,Z 1269.091,A -85,B 0,C 180,E1 31291.953,E2 31291.953} C_VEL
LIN {X 0,Y 188.485,Z 1242.055,A -85,B 0,C 180,E1 31310.273,E2 31310.273} C_VEL
LIN {X 0,Y 256.939,Z 1201.311,A -85,B 0,C 180,E1 31318.567,E2 31318.567} C_VEL
LIN {X 0,Y 275.821,Z 1187.263,A -85,B 0,C 180,E1 31320.297,E2 31320.297} C_VEL
LIN {X 0,Y 209.021,Z 1230.895,A -85,B 0,C 180,E1 31327.101,E2 31327.101} C_VEL
LIN {X 0,Y 142.355,Z 1261.326,A -85,B 0,C 180,E1 31341.228,E2 31341.228} C_VEL
LIN {X 0,Y 94.933,Z 1277.107,A -85,B 0,C 180,E1 31370.284,E2 31370.284} C_VEL
LIN {X 0,Y 82.837,Z 1280.939,A -85,B 0,C 180,E1 31404.748,E2 31404.748} C_VEL
LIN {X 0,Y 86.831,Z 1279.484,A -85,B 0,C 180,E1 31435.89,E2 31435.89} C_VEL
LIN {X 0,Y 127.602,Z 1266.582,A -85,B 0,C 180,E1 31473.046,E2 31473.046} C_VEL
LIN {X 0,Y 192.319,Z 1239.485,A -85,B 0,C 180,E1 31490.297,E2 31490.297} C_VEL
LIN {X 0,Y 234.416,Z 1216,A -85,B 0,C 180,E1 31495.892,E2 31495.892} C_VEL
LIN {X 0,Y 250.199,Z 1205.689,A -85,B 0,C 180,E1 31499.406,E2 31499.406} C_VEL
LIN {X 0,Y 253.061,Z 1203.699,A -85,B 0,C 180,E1 31499.875,E2 31499.875} C_VEL
LIN {X 0,Y 183.176,Z 1243.84,A -85,B 0,C 180,E1 31507.841,E2 31507.841} C_VEL
LIN {X 0,Y 117.77,Z 1269.682,A -85,B 0,C 180,E1 31525.535,E2 31525.535} C_VEL
LIN {X 0,Y 79.241,Z 1281.104,A -85,B 0,C 180,E1 31561.415,E2 31561.415} C_VEL
LIN {X 0,Y 74.733,Z 1282.654,A -85,B 0,C 180,E1 31595.823,E2 31595.823} C_VEL
LIN {X 0,Y 92.375,Z 1277.384,A -85,B 0,C 180,E1 31637.626,E2 31637.626} C_VEL
LIN {X 0,Y 153.248,Z 1256.977,A -85,B 0,C 180,E1 31666.099,E2 31666.099} C_VEL
LIN {X 0,Y 223.024,Z 1222.898,A -85,B 0,C 180,E1 31677.324,E2 31677.324} C_VEL
LIN {X 0,Y 252.896,Z 1204.006,A -85,B 0,C 180,E1 31680.322,E2 31680.322} C_VEL
LIN {X 0,Y 183.903,Z 1243.167,A -85,B 0,C 180,E1 31688.286,E2 31688.286} C_VEL
LIN {X 0,Y 118.916,Z 1268.413,A -85,B 0,C 180,E1 31705.721,E2 31705.721} C_VEL
LIN {X 0,Y 79.509,Z 1279.599,A -85,B 0,C 180,E1 31741.521,E2 31741.521} C_VEL
LIN {X 0,Y 74.996,Z 1281.017,A -85,B 0,C 180,E1 31775.804,E2 31775.804} C_VEL
LIN {X 0,Y 92.794,Z 1275.968,A -85,B 0,C 180,E1 31817.345,E2 31817.345} C_VEL
LIN {X 0,Y 153.198,Z 1256.193,A -85,B 0,C 180,E1 31845.572,E2 31845.572} C_VEL
LIN {X 0,Y 224.023,Z 1221.972,A -85,B 0,C 180,E1 31856.876,E2 31856.876} C_VEL
LIN {X 0,Y 250.199,Z 1205.689,A -85,B 0,C 180,E1 31859.406,E2 31859.406} C_VEL
LIN {X 0,Y 220.093,Z 1224.217,A -85,B 0,C 180,E1 31860.801,E2 31860.801} C_VEL
LIN {X 0,Y 148.885,Z 1257.783,A -85,B 0,C 180,E1 31871.34,E2 31871.34} C_VEL
LIN {X 0,Y 86.987,Z 1277.253,A -85,B 0,C 180,E1 31898.322,E2 31898.322} C_VEL
LIN {X 0,Y 66.776,Z 1282.561,A -85,B 0,C 180,E1 31943.479,E2 31943.479} C_VEL
LIN {X 0,Y 72.196,Z 1281.032,A -85,B 0,C 180,E1 31981.677,E2 31981.677} C_VEL
LIN {X 0,Y 120.532,Z 1267.726,A -85,B 0,C 180,E1 32020.673,E2 32020.673} C_VEL
LIN {X 0,Y 190.069,Z 1240.121,A -85,B 0,C 180,E1 32035.83,E2 32035.83} C_VEL
LIN {X 0,Y 229.737,Z 1218.787,A -85,B 0,C 180,E1 32040.309,E2 32040.309} C_VEL
LIN {X 0,Y 161.359,Z 1252.589,A -85,B 0,C 180,E1 32049.306,E2 32049.306} C_VEL
LIN {X 0,Y 97.431,Z 1273.625,A -85,B 0,C 180,E1 32071.121,E2 32071.121} C_VEL
LIN {X 0,Y 68.337,Z 1280.69,A -85,B 0,C 180,E1 32110.557,E2 32110.557} C_VEL
LIN {X 0,Y 66.996,Z 1281.105,A -85,B 0,C 180,E1 32136.499,E2 32136.499} C_VEL
LIN {X 0,Y 90.223,Z 1275.351,A -85,B 0,C 180,E1 32183.756,E2 32183.756} C_VEL
LIN {X 0,Y 151.327,Z 1256.285,A -85,B 0,C 180,E1 32208.647,E2 32208.647} C_VEL
LIN {X 0,Y 223.547,Z 1222.166,A -85,B 0,C 180,E1 32218.993,E2 32218.993} C_VEL
LIN {X 0,Y 231.383,Z 1217.687,A -85,B 0,C 180,E1 32219.759,E2 32219.759} C_VEL
LIN {X 0,Y 220.093,Z 1224.217,A -85,B 0,C 180,E1 32220.801,E2 32220.801} C_VEL
LIN {X 0,Y 202.431,Z 1233.584,A -85,B 0,C 180,E1 32219.196,E2 32219.196} C_VEL
LIN {X 0,Y 199.821,Z 1234.919,A -85,B 0,C 180,E1 32218.859,E2 32218.859} C_VEL
LIN {X 0,Y 127.125,Z 1264.228,A -85,B 0,C 180,E1 32206.445,E2 32206.445} C_VEL
LIN {X 0,Y 73.072,Z 1278.181,A -85,B 0,C 180,E1 32176.586,E2 32176.586} C_VEL
LIN {X 0,Y 58.983,Z 1281.194,A -85,B 0,C 180,E1 32137.387,E2 32137.387} C_VEL
LIN {X 0,Y 66.093,Z 1279.703,A -85,B 0,C 180,E1 32093.811,E2 32093.811} C_VEL
LIN {X 0,Y 118.362,Z 1266.938,A -85,B 0,C 180,E1 32056.066,E2 32056.066} C_VEL
LIN {X 0,Y 189.698,Z 1239.896,A -85,B 0,C 180,E1 32042.136,E2 32042.136} C_VEL
LIN {X 0,Y 204.732,Z 1232.556,A -85,B 0,C 180,E1 32039.982,E2 32039.982} C_VEL
LIN {X 0,Y 131.627,Z 1263.321,A -85,B 0,C 180,E1 32028.328,E2 32028.328} C_VEL
LIN {X 0,Y 72.725,Z 1279.309,A -85,B 0,C 180,E1 31996.874,E2 31996.874} C_VEL
LIN {X 0,Y 58.724,Z 1282.477,A -85,B 0,C 180,E1 31957.418,E2 31957.418} C_VEL
LIN {X 0,Y 65.963,Z 1280.814,A -85,B 0,C 180,E1 31913.245,E2 31913.245} C_VEL
LIN {X 0,Y 118.066,Z 1267.57,A -85,B 0,C 180,E1 31875.556,E2 31875.556} C_VEL
LIN {X 0,Y 189.645,Z 1239.906,A -85,B 0,C 180,E1 31861.631,E2 31861.631} C_VEL
LIN {X 0,Y 208.149,Z 1230.646,A -85,B 0,C 180,E1 31859.715,E2 31859.715} C_VEL
LIN {X 0,Y 199.821,Z 1234.919,A -85,B 0,C 180,E1 31858.859,E2 31858.859} C_VEL
LIN {X 0,Y 167.588,Z 1249.358,A -85,B 0,C 180,E1 31857.758,E2 31857.758} C_VEL
LIN {X 0,Y 94.937,Z 1272.523,A -85,B 0,C 180,E1 31840.332,E2 31840.332} C_VEL
LIN {X 0,Y 53.347,Z 1280.844,A -85,B 0,C 180,E1 31795.241,E2 31795.241} C_VEL
LIN {X 0,Y 50.832,Z 1281.291,A -85,B 0,C 180,E1 31761.422,E2 31761.422} C_VEL
LIN {X 0,Y 83.889,Z 1275.105,A -85,B 0,C 180,E1 31705.327,E2 31705.327} C_VEL
LIN {X 0,Y 155.807,Z 1254.104,A -85,B 0,C 180,E1 31683.913,E2 31683.913} C_VEL
LIN {X 0,Y 183.452,Z 1242.77,A -85,B 0,C 180,E1 31680.257,E2 31680.257} C_VEL
LIN {X 0,Y 109.205,Z 1269.499,A -85,B 0,C 180,E1 31666.432,E2 31666.432} C_VEL
LIN {X 0,Y 58.898,Z 1280.853,A -85,B 0,C 180,E1 31630.068,E2 31630.068} C_VEL
LIN {X 0,Y 50.787,Z 1282.384,A -85,B 0,C 180,E1 31581.413,E2 31581.413} C_VEL
LIN {X 0,Y 83.574,Z 1275.835,A -85,B 0,C 180,E1 31524.864,E2 31524.864} C_VEL
LIN {X 0,Y 155.708,Z 1254.215,A -85,B 0,C 180,E1 31503.328,E2 31503.328} C_VEL
LIN {X 0,Y 183.743,Z 1242.507,A -85,B 0,C 180,E1 31499.687,E2 31499.687} C_VEL
LIN {X 0,Y 167.588,Z 1249.358,A -85,B 0,C 180,E1 31497.758,E2 31497.758} C_VEL
LIN {X 0,Y 134.493,Z 1261.248,A -85,B 0,C 180,E1 31495.942,E2 31495.942} C_VEL
LIN {X 0,Y 67.914,Z 1277.605,A -85,B 0,C 180,E1 31471.906,E2 31471.906} C_VEL
LIN {X 0,Y 43.013,Z 1281.371,A -85,B 0,C 180,E1 31420.155,E2 31420.155} C_VEL
LIN {X 0,Y 53.129,Z 1279.955,A -85,B 0,C 180,E1 31364.472,E2 31364.472} C_VEL
LIN {X 0,Y 114.858,Z 1267.12,A -85,B 0,C 180,E1 31328.004,E2 31328.004} C_VEL
LIN {X 0,Y 159.237,Z 1252.863,A -85,B 0,C 180,E1 31320.254,E2 31320.254} C_VEL
LIN {X 0,Y 86.932,Z 1274.438,A -85,B 0,C 180,E1 31303.632,E2 31303.632} C_VEL
LIN {X 0,Y 45.909,Z 1281.828,A -85,B 0,C 180,E1 31259.702,E2 31259.702} C_VEL
LIN {X 0,Y 42.812,Z 1282.296,A -85,B 0,C 180,E1 31219.797,E2 31219.797} C_VEL
LIN {X 0,Y 80.427,Z 1275.744,A -85,B 0,C 180,E1 31159.47,E2 31159.47} C_VEL
LIN {X 0,Y 155.447,Z 1254.122,A -85,B 0,C 180,E1 31140.222,E2 31140.222} C_VEL
LIN {X 0,Y 159.24,Z 1252.748,A -85,B 0,C 180,E1 31139.662,E2 31139.662} C_VEL
LIN {X 0,Y 134.493,Z 1261.248,A -85,B 0,C 180,E1 31135.942,E2 31135.942} C_VEL
LIN {X 0,Y 100.666,Z 1270.518,A -85,B 0,C 180,E1 31133.087,E2 31133.087} C_VEL
LIN {X 0,Y 47.756,Z 1280.022,A -85,B 0,C 180,E1 31102.553,E2 31102.553} C_VEL
LIN {X 0,Y 34.948,Z 1281.468,A -85,B 0,C 180,E1 31037.47,E2 31037.47} C_VEL
LIN {X 0,Y 78.252,Z 1275.285,A -85,B 0,C 180,E1 30974.304,E2 30974.304} C_VEL
LIN {X 0,Y 135.15,Z 1261.134,A -85,B 0,C 180,E1 30960.246,E2 30960.246} C_VEL
LIN {X 0,Y 65.9,Z 1277.959,A -85,B 0,C 180,E1 30940.027,E2 30940.027} C_VEL
LIN {X 0,Y 34.856,Z 1282.213,A -85,B 0,C 180,E1 30882.563,E2 30882.563} C_VEL
LIN {X 0,Y 47.484,Z 1280.654,A -85,B 0,C 180,E1 30817.017,E2 30817.017} C_VEL
LIN {X 0,Y 117.644,Z 1266.317,A -85,B 0,C 180,E1 30782.577,E2 30782.577} C_VEL
LIN {X 0,Y 135.317,Z 1260.994,A -85,B 0,C 180,E1 30779.707,E2 30779.707} C_VEL
LIN {X 0,Y 100.666,Z 1270.518,A -85,B 0,C 180,E1 30773.087,E2 30773.087} C_VEL
LIN {X 0,Y 66.527,Z 1277.019,A -85,B 0,C 180,E1 30767.821,E2 30767.821} C_VEL
LIN {X 0,Y 27.246,Z 1281.548,A -85,B 0,C 180,E1 30706.161,E2 30706.161} C_VEL
LIN {X 0,Y 43.245,Z 1280.134,A -85,B 0,C 180,E1 30628.755,E2 30628.755} C_VEL
LIN {X 0,Y 109.531,Z 1268.357,A -85,B 0,C 180,E1 30600.309,E2 30600.309} C_VEL
LIN {X 0,Y 43.05,Z 1280.584,A -85,B 0,C 180,E1 30571.724,E2 30571.724} C_VEL
LIN {X 0,Y 27.038,Z 1282.118,A -85,B 0,C 180,E1 30493.712,E2 30493.712} C_VEL
LIN {X 0,Y 76.499,Z 1275.56,A -85,B 0,C 180,E1 30427.599,E2 30427.599} C_VEL
LIN {X 0,Y 110.125,Z 1268.133,A -85,B 0,C 180,E1 30419.647,E2 30419.647} C_VEL
LIN {X 0,Y 66.527,Z 1277.019,A -85,B 0,C 180,E1 30407.821,E2 30407.821} C_VEL
LIN {X 0,Y 33.011,Z 1280.739,A -85,B 0,C 180,E1 30394.386,E2 30394.386} C_VEL
LIN {X 0,Y 19.493,Z 1281.645,A -85,B 0,C 180,E1 30307.11,E2 30307.11} C_VEL
LIN {X 0,Y 75.875,Z 1275.466,A -85,B 0,C 180,E1 30242.067,E2 30242.067} C_VEL
LIN {X 0,Y 82.229,Z 1274.412,A -85,B 0,C 180,E1 30240.171,E2 30240.171} C_VEL
LIN {X 0,Y 27.478,Z 1281.562,A -85,B 0,C 180,E1 30205.876,E2 30205.876} C_VEL
LIN {X 0,Y 19.414,Z 1282.03,A -85,B 0,C 180,E1 30127.007,E2 30127.007} C_VEL
LIN {X 0,Y 75.848,Z 1275.468,A -85,B 0,C 180,E1 30061.329,E2 30061.329} C_VEL
LIN {X 0,Y 82.269,Z 1274.345,A -85,B 0,C 180,E1 30059.829,E2 30059.829} C_VEL
LIN {X 0,Y 33.011,Z 1280.739,A -85,B 0,C 180,E1 30034.386,E2 30034.386} C_VEL
LIN {X 0,Y 11.466,Z 1281.732,A -85,B 0,C 180,E1 29939.524,E2 29939.524} C_VEL
LIN {X 0,Y 53.078,Z 1278.768,A -85,B 0,C 180,E1 29879.922,E2 29879.922} C_VEL
LIN {X 0,Y 12.354,Z 1281.947,A -85,B 0,C 180,E1 29827.859,E2 29827.859} C_VEL
LIN {X 0,Y 23.865,Z 1281.452,A -85,B 0,C 180,E1 29717.595,E2 29717.595} C_VEL
LIN {X 0,Y 53.085,Z 1278.725,A -85,B 0,C 180,E1 29699.198,E2 29699.198} C_VEL
LIN {X 0,Y 12.536,Z 1281.725,A -85,B 0,C 180,E1 29647.224,E2 29647.224} C_VEL
LIN {X 0,Y 11.466,Z 1281.732,A -85,B 0,C 180,E1 29579.524,E2 29579.524} C_VEL
LIN {X 0,Y 7.665,Z 1281.842,A -85,B 0,C 180,E1 29696.43,E2 29696.43} C_VEL
LIN {X 0,Y 15.66,Z 1281.655,A -85,B 0,C 180,E1 29701.254,E2 29701.254} C_VEL
LIN {X 0,Y 18.769,Z 1281.578,A -85,B 0,C 180,E1 29699.498,E2 29699.498} C_VEL
LIN {X 0,Y 18.418,Z 1281.594,A -85,B 0,C 180,E1 29520.41,E2 29520.41} C_VEL
LIN {X 0,Y 15.66,Z 1281.655,A -85,B 0,C 180,E1 29341.254,E2 29341.254} C_VEL
LIN {X 0,Y 17.678,Z 1283.654,A -85,B 0,C 180,E1 29340.043,E2 29340.043} C_VEL
LIN {X 0,Y 17.678,Z 1292,A -85,B 0,C 180,E1 29340.043,E2 29340.043} C_VEL
LIN {X 0,Y 17.678,Z 1292,A -85,B 0,C 180,E1 29340.043,E2 29340.043}

QRS_NEXT_CUT()
PTP {E1 29337.209,E2 29337.209}
PTP {X 0,Y 759.904,A -85,B 0,C 180,E1 29337.209,E2 29337.209,E3 0,E4 0,E5 0,E6 0}
QRS_SPEED_INIT()
LIN {X 0,Y 759.904,Z 1292,A -85,B 0,C 180,E1 29337.209,E2 29337.209,E3 0,E4 0,E5 0,E6 0} C_VEL
LIN {X 0,Y 759.904,Z 406.645,A -85,B 0,C 180,E1 29337.209,E2 29337.209} C_VEL
LIN {X 0,Y 759.904,Z 398.565,A -85,B 0,C 180,E1 29337.209,E2 29337.209} C_VEL
LIN {X 0,Y 759.909,Z 396.565,A -85,B 0,C 180,E1 29337.059,E2 29337.059} C_VEL
LIN {X 0,Y 759.875,Z 396.57,A -85,B 0,C 180,E1 29334.26,E2 29334.26} C_VEL
LIN {X 0,Y 759.911,Z 396.575,A -85,B 0,C 180,E1 29331.449,E2 29331.449} C_VEL
LIN {X 0,Y 759.902,Z 396.565,A -85,B 0,C 180,E1 29328.463,E2 29328.463} C_VEL
LIN {X 0,Y 759.909,Z 396.576,A -85,B 0,C 180,E1 29325.522,E2 29325.522} C_VEL
LIN {X 0,Y 759.907,Z 396.565,A -85,B 0,C 180,E1 29322.542,E2 29322.542} C_VEL
LIN {X 0,Y 759.892,Z 396.572,A -85,B 0,C 180,E1 29319.673,E2 29319.673} C_VEL
LIN {X 0,Y 759.889,Z 396.572,A -85,B 0,C 180,E1 29316.891,E2 29316.891} C_VEL
LIN {X 0,Y 759.908,Z 396.564,A -85,B 0,C 180,E1 29314.013,E2 29314.013} C_VEL
LIN {X 0,Y 759.904,Z 396.575,A -85,B 0,C 180,E1 29311.039,E2 29311.039} C_VEL
LIN {X 0,Y 759.895,Z 396.566,A -85,B 0,C 180,E1 29308.153,E2 29308.153} C_VEL
LIN {X 0,Y 759.91,Z 396.575,A -85,B 0,C 180,E1 29305.176,E2 29305.176} C_VEL
LIN {X 0,Y 759.871,Z 396.57,A -85,B 0,C 180,E1 29302.387,E2 29302.387} C_VEL
LIN {X 0,Y 759.918,Z 396.565,A -85,B 0,C 180,E1 29299.627,E2 29299.627} C_VEL
LIN {X 0,Y 759.889,Z 396.576,A -85,B 0,C 180,E1 29296.691,E2 29296.691} C_VEL
LIN {X 0,Y 759.865,Z 396.571,A -85,B 0,C 180,E1 29293.963,E2 29293.963} C_VEL
LIN {X 0,Y 759.861,Z 396.582,A -85,B 0,C 180,E1 29292.281,E2 29292.281} C_VEL
LIN {X 0,Y 759.916,Z 418.206,A -85,B 0,C 180,E1 29290.865,E2 29290.865} C_VEL
LIN {X 0,Y 759.911,Z 630.685,A -85,B 0,C 180,E1 29288.311,E2 29288.311} C_VEL
LIN {X 0,Y 759.915,Z 855.958,A -85,B 0,C 180,E1 29285.698,E2 29285.698} C_VEL
LIN {X 0,Y 759.919,Z 897.834,A -85,B 0,C 180,E1 29285.192,E2 29285.192} C_VEL
LIN {X 0,Y 759.907,Z 923.235,A -85,B 0,C 180,E1 29284.752,E2 29284.752} C_VEL
LIN {X 0,Y 759.908,Z 950.602,A -85,B 0,C 180,E1 29284.118,E2 29284.118} C_VEL
LIN {X 0,Y 759.908,Z 973.25,A -85,B 0,C 180,E1 29283.458,E2 29283.458} C_VEL
LIN {X 0,Y 759.918,Z 993.524,A -85,B 0,C 180,E1 29282.776,E2 29282.776} C_VEL
LIN {X 0,Y 759.917,Z 1018.316,A -85,B 0,C 180,E1 29281.817,E2 29281.817} C_VEL
LIN {X 0,Y 759.909,Z 1042.789,A -85,B 0,C 180,E1 29280.7,E2 29280.7} C_VEL
LIN {X 0,Y 759.913,Z 1061.867,A -85,B 0,C 180,E1 29279.723,E2 29279.723} C_VEL
LIN {X 0,Y 759.904,Z 1079.91,A -85,B 0,C 180,E1 29278.704,E2 29278.704} C_VEL
LIN {X 0,Y 759.907,Z 1099.133,A -85,B 0,C 180,E1 29277.507,E2 29277.507} C_VEL
LIN {X 0,Y 759.895,Z 1122.116,A -85,B 0,C 180,E1 29275.904,E2 29275.904} C_VEL
LIN {X 0,Y 759.916,Z 1139.739,A -85,B 0,C 180,E1 29274.529,E2 29274.529} C_VEL
LIN {X 0,Y 759.905,Z 1157.505,A -85,B 0,C 180,E1 29273.005,E2 29273.005} C_VEL
LIN {X 0,Y 759.906,Z 1176.041,A -85,B 0,C 180,E1 29271.215,E2 29271.215} C_VEL
LIN {X 0,Y 759.88,Z 1189.541,A -85,B 0,C 180,E1 29269.767,E2 29269.767} C_VEL
LIN {X 0,Y 759.905,Z 1202.35,A -85,B 0,C 180,E1 29268.251,E2 29268.251} C_VEL
LIN {X 0,Y 759.903,Z 1216.276,A -85,B 0,C 180,E1 29266.416,E2 29266.416} C_VEL
LIN {X 0,Y 759.917,Z 1228.913,A -85,B 0,C 180,E1 29264.479,E2 29264.479} C_VEL
LIN {X 0,Y 759.899,Z 1238.319,A -85,B 0,C 180,E1 29262.831,E2 29262.831} C_VEL
LIN {X 0,Y 759.911,Z 1246.28,A -85,B 0,C 180,E1 29261.231,E2 29261.231} C_VEL
LIN {X 0,Y 759.889,Z 1252.854,A -85,B 0,C 180,E1 29259.698,E2 29259.698} C_VEL
LIN {X 0,Y 759.892,Z 1258.913,A -85,B 0,C 180,E1 29258.019,E2 29258.019} C_VEL
LIN {X 0,Y 759.915,Z 1264.422,A -85,B 0,C 180,E1 29256.12,E2 29256.12} C_VEL
LIN {X 0,Y 759.916,Z 1268.6,A -85,B 0,C 180,E1 29254.076,E2 29254.076} C_VEL
LIN {X 0,Y 759.908,Z 1270.836,A -85,B 0,C 180,E1 29252.264,E2 29252.264} C_VEL
LIN {X 0,Y 759.866,Z 1271.791,A -85,B 0,C 180,E1 29250.681,E2 29250.681} C_VEL
LIN {X 0,Y 759.863,Z 1271.774,A -85,B 0,C 180,E1 29249.173,E2 29249.173} C_VEL
LIN {X 0,Y 759.901,Z 1270.785,A -85,B 0,C 180,E1 29247.589,E2 29247.589} C_VEL
LIN {X 0,Y 759.919,Z 1268.507,A -85,B 0,C 180,E1 29245.777,E2 29245.777} C_VEL
LIN {X 0,Y 759.916,Z 1264.47,A -85,B 0,C 180,E1 29243.809,E2 29243.809} C_VEL
LIN {X 0,Y 759.9,Z 1258.974,A -85,B 0,C 180,E1 29241.909,E2 29241.909} C_VEL
LIN {X 0,Y 759.887,Z 1252.926,A -85,B 0,C 180,E1 29240.23,E2 29240.23} C_VEL
LIN {X 0,Y 759.907,Z 1246.362,A -85,B 0,C 180,E1 29238.696,E2 29238.696} C_VEL
LIN {X 0,Y 759.911,Z 1238.721,A -85,B 0,C 180,E1 29237.155,E2 29237.155} C_VEL
LIN {X 0,Y 759.917,Z 1229.708,A -85,B 0,C 180,E1 29235.564,E2 29235.564} C_VEL
LIN {X 0,Y 759.888,Z 1218.735,A -85,B 0,C 180,E1 29233.856,E2 29233.856} C_VEL
LIN {X 0,Y 759.911,Z 1203.556,A -85,B 0,C 180,E1 29231.807,E2 29231.807} C_VEL
LIN {X 0,Y 759.88,Z 1190.38,A -85,B 0,C 180,E1 29230.238,E2 29230.238} C_VEL
LIN {X 0,Y 759.901,Z 1176.954,A -85,B 0,C 180,E1 29228.79,E2 29228.79} C_VEL
LIN {X 0,Y 759.907,Z 1159.494,A -85,B 0,C 180,E1 29227.081,E2 29227.081} C_VEL
LIN {X 0,Y 759.911,Z 1140.392,A -85,B 0,C 180,E1 29225.434,E2 29225.434} C_VEL
LIN {X 0,Y 759.898,Z 1123.369,A -85,B 0,C 180,E1 29224.101,E2 29224.101} C_VEL
LIN {X 0,Y 759.918,Z 1101.937,A -85,B 0,C 180,E1 29222.583,E2 29222.583} C_VEL
LIN {X 0,Y 759.908,Z 1080.79,A -85,B 0,C 180,E1 29221.258,E2 29221.258} C_VEL
LIN {X 0,Y 759.912,Z 1062.51,A -85,B 0,C 180,E1 29220.221,E2 29220.221} C_VEL
LIN {X 0,Y 759.912,Z 1043.948,A -85,B 0,C 180,E1 29219.267,E2 29219.267} C_VEL
LIN {X 0,Y 759.915,Z 1023.797,A -85,B 0,C 180,E1 29218.336,E2 29218.336} C_VEL
LIN {X 0,Y 759.917,Z 998.576,A -85,B 0,C 180,E1 29217.312,E2 29217.312} C_VEL
LIN {X 0,Y 759.907,Z 974.687,A -85,B 0,C 180,E1 29216.496,E2 29216.496} C_VEL
LIN {X 0,Y 759.907,Z 951.7,A -85,B 0,C 180,E1 29215.821,E2 29215.821} C_VEL
LIN {X 0,Y 759.907,Z 924.838,A -85,B 0,C 180,E1 29215.192,E2 29215.192} C_VEL
LIN {X 0,Y 759.914,Z 899.343,A -85,B 0,C 180,E1 29214.739,E2 29214.739} C_VEL
LIN {X 0,Y 759.916,Z 860.767,A -85,B 0,C 180,E1 29214.267,E2 29214.267} C_VEL
LIN {X 0,Y 759.91,Z 637.415,A -85,B 0,C 180,E1 29211.678,E2 29211.678} C_VEL
LIN {X 0,Y 759.907,Z 427.04,A -85,B 0,C 180,E1 29209.152,E2 29209.152} C_VEL
LIN {X 0,Y 759.913,Z 417.662,A -85,B 0,C 180,E1 29209.028,E2 29209.028} C_VEL
LIN {X 0,Y 759.851,Z 396.579,A -85,B 0,C 180,E1 29207.615,E2 29207.615} C_VEL
LIN {X 0,Y 759.918,Z 396.577,A -85,B 0,C 180,E1 29204.942,E2 29204.942} C_VEL
LIN {X 0,Y 759.86,Z 396.57,A -85,B 0,C 180,E1 29201.978,E2 29201.978} C_VEL
LIN {X 0,Y 759.843,Z 396.573,A -85,B 0,C 180,E1 29199.464,E2 29199.464} C_VEL
LIN {X 0,Y 759.881,Z 396.576,A -85,B 0,C 180,E1 29196.872,E2 29196.872} C_VEL
LIN {X 0,Y 759.87,Z 396.569,A -85,B 0,C 180,E1 29193.822,E2 29193.822} C_VEL
LIN {X 0,Y 759.84,Z 396.572,A -85,B 0,C 180,E1 29191.318,E2 29191.318} C_VEL
LIN {X 0,Y 759.848,Z 396.574,A -85,B 0,C 180,E1 29188.878,E2 29188.878} C_VEL
LIN {X 0,Y 759.914,Z 396.574,A -85,B 0,C 180,E1 29186.154,E2 29186.154} C_VEL
LIN {X 0,Y 759.851,Z 396.571,A -85,B 0,C 180,E1 29183.304,E2 29183.304} C_VEL
LIN {X 0,Y 759.835,Z 396.572,A -85,B 0,C 180,E1 29180.893,E2 29180.893} C_VEL
LIN {X 0,Y 759.845,Z 396.574,A -85,B 0,C 180,E1 29178.49,E2 29178.49} C_VEL
LIN {X 0,Y 759.915,Z 396.573,A -85,B 0,C 180,E1 29175.727,E2 29175.727} C_VEL
LIN {X 0,Y 759.846,Z 396.572,A -85,B 0,C 180,E1 29172.927,E2 29172.927} C_VEL
LIN {X 0,Y 759.831,Z 396.573,A -85,B 0,C 180,E1 29170.54,E2 29170.54} C_VEL
LIN {X 0,Y 759.837,Z 396.573,A -85,B 0,C 180,E1 29168.171,E2 29168.171} C_VEL
LIN {X 0,Y 759.919,Z 396.576,A -85,B 0,C 180,E1 29165.436,E2 29165.436} C_VEL
LIN {X 0,Y 759.842,Z 396.571,A -85,B 0,C 180,E1 29162.564,E2 29162.564} C_VEL
LIN {X 0,Y 759.827,Z 396.574,A -85,B 0,C 180,E1 29160.226,E2 29160.226} C_VEL
LIN {X 0,Y 759.828,Z 396.574,A -85,B 0,C 180,E1 29157.888,E2 29157.888} C_VEL
LIN {X 0,Y 759.864,Z 396.575,A -85,B 0,C 180,E1 29155.396,E2 29155.396} C_VEL
LIN {X 0,Y 759.854,Z 396.572,A -85,B 0,C 180,E1 29152.362,E2 29152.362} C_VEL
LIN {X 0,Y 759.824,Z 396.573,A -85,B 0,C 180,E1 29149.92,E2 29149.92} C_VEL
LIN {X 0,Y 759.821,Z 396.575,A -85,B 0,C 180,E1 29147.614,E2 29147.614} C_VEL
LIN {X 0,Y 759.834,Z 396.575,A -85,B 0,C 180,E1 29145.268,E2 29145.268} C_VEL
LIN {X 0,Y 759.919,Z 396.573,A -85,B 0,C 180,E1 29142.463,E2 29142.463} C_VEL
LIN {X 0,Y 759.83,Z 396.573,A -85,B 0,C 180,E1 29139.748,E2 29139.748} C_VEL
LIN {X 0,Y 759.818,Z 396.575,A -85,B 0,C 180,E1 29137.476,E2 29137.476} C_VEL
LIN {X 0,Y 759.815,Z 396.575,A -85,B 0,C 180,E1 29135.221,E2 29135.221} C_VEL
LIN {X 0,Y 759.822,Z 396.576,A -85,B 0,C 180,E1 29132.914,E2 29132.914} C_VEL
LIN {X 0,Y 759.878,Z 396.577,A -85,B 0,C 180,E1 29130.346,E2 29130.346} C_VEL
LIN {X 0,Y 759.837,Z 396.575,A -85,B 0,C 180,E1 29127.438,E2 29127.438} C_VEL
LIN {X 0,Y 759.814,Z 396.575,A -85,B 0,C 180,E1 29125.079,E2 29125.079} C_VEL
LIN {X 0,Y 759.809,Z 396.576,A -85,B 0,C 180,E1 29122.84,E2 29122.84} C_VEL
LIN {X 0,Y 759.809,Z 396.577,A -85,B 0,C 180,E1 29120.632,E2 29120.632} C_VEL
LIN {X 0,Y 759.812,Z 396.576,A -85,B 0,C 180,E1 29118.452,E2 29118.452} C_VEL
LIN {X 0,Y 759.848,Z 396.578,A -85,B 0,C 180,E1 29115.988,E2 29115.988} C_VEL
LIN {X 0,Y 759.831,Z 396.603,A -85,B 0,C 180,E1 29112.948,E2 29112.948} C_VEL
LIN {X 0,Y 759.867,Z 427.769,A -85,B 0,C 180,E1 29110.919,E2 29110.919} C_VEL
LIN {X 0,Y 759.909,Z 624.729,A -85,B 0,C 180,E1 29108.545,E2 29108.545} C_VEL
LIN {X 0,Y 759.908,Z 844.308,A -85,B 0,C 180,E1 29105.99,E2 29105.99} C_VEL
LIN {X 0,Y 759.913,Z 906.257,A -85,B 0,C 180,E1 29105.261,E2 29105.261} C_VEL
LIN {X 0,Y 759.907,Z 932.692,A -85,B 0,C 180,E1 29104.808,E2 29104.808} C_VEL
LIN {X 0,Y 759.908,Z 959.959,A -85,B 0,C 180,E1 29104.179,E2 29104.179} C_VEL
LIN {X 0,Y 759.91,Z 981.947,A -85,B 0,C 180,E1 29103.544,E2 29103.544} C_VEL
LIN {X 0,Y 759.919,Z 999.626,A -85,B 0,C 180,E1 29102.959,E2 29102.959} C_VEL
LIN {X 0,Y 759.918,Z 1017.676,A -85,B 0,C 180,E1 29102.286,E2 29102.286} C_VEL
LIN {X 0,Y 759.913,Z 1036.762,A -85,B 0,C 180,E1 29101.487,E2 29101.487} C_VEL
LIN {X 0,Y 759.912,Z 1055.586,A -85,B 0,C 180,E1 29100.607,E2 29100.607} C_VEL
LIN {X 0,Y 759.911,Z 1074.087,A -85,B 0,C 180,E1 29099.649,E2 29099.649} C_VEL
LIN {X 0,Y 759.906,Z 1094.427,A -85,B 0,C 180,E1 29098.482,E2 29098.482} C_VEL
LIN {X 0,Y 759.913,Z 1117.461,A -85,B 0,C 180,E1 29096.993,E2 29096.993} C_VEL
LIN {X 0,Y 759.904,Z 1134.989,A -85,B 0,C 180,E1 29095.732,E2 29095.732} C_VEL
LIN {X 0,Y 759.899,Z 1152.38,A -85,B 0,C 180,E1 29094.359,E2 29094.359} C_VEL
LIN {X 0,Y 759.915,Z 1173.1,A -85,B 0,C 180,E1 29092.528,E2 29092.528} C_VEL
LIN {X 0,Y 759.902,Z 1188.08,A -85,B 0,C 180,E1 29091.049,E2 29091.049} C_VEL
LIN {X 0,Y 759.887,Z 1202.113,A -85,B 0,C 180,E1 29089.522,E2 29089.522} C_VEL
LIN {X 0,Y 759.883,Z 1217.773,A -85,B 0,C 180,E1 29087.613,E2 29087.613} C_VEL
LIN {X 0,Y 759.884,Z 1230.263,A -85,B 0,C 180,E1 29085.869,E2 29085.869} C_VEL
LIN {X 0,Y 759.914,Z 1240.14,A -85,B 0,C 180,E1 29084.319,E2 29084.319} C_VEL
LIN {X 0,Y 759.912,Z 1248.892,A -85,B 0,C 180,E1 29082.768,E2 29082.768} C_VEL
LIN {X 0,Y 759.906,Z 1256.51,A -85,B 0,C 180,E1 29081.227,E2 29081.227} C_VEL
LIN {X 0,Y 759.877,Z 1263.358,A -85,B 0,C 180,E1 29079.617,E2 29079.617} C_VEL
LIN {X 0,Y 759.882,Z 1270.36,A -85,B 0,C 180,E1 29077.635,E2 29077.635} C_VEL
LIN {X 0,Y 759.914,Z 1275.598,A -85,B 0,C 180,E1 29075.661,E2 29075.661} C_VEL
LIN {X 0,Y 759.912,Z 1279.283,A -85,B 0,C 180,E1 29073.694,E2 29073.694} C_VEL
LIN {X 0,Y 759.913,Z 1281.55,A -85,B 0,C 180,E1 29071.506,E2 29071.506} C_VEL
LIN {X 0,Y 759.869,Z 1281.871,A -85,B 0,C 180,E1 29069.545,E2 29069.545} C_VEL
LIN {X 0,Y 759.913,Z 1281.011,A -85,B 0,C 180,E1 29067.887,E2 29067.887} C_VEL
LIN {X 0,Y 759.911,Z 1278.925,A -85,B 0,C 180,E1 29066.075,E2 29066.075} C_VEL
LIN {X 0,Y 759.913,Z 1274.73,A -85,B 0,C 180,E1 29063.956,E2 29063.956} C_VEL
LIN {X 0,Y 759.888,Z 1269.32,A -85,B 0,C 180,E1 29062.057,E2 29062.057} C_VEL
LIN {X 0,Y 759.884,Z 1263.035,A -85,B 0,C 180,E1 29060.302,E2 29060.302} C_VEL
LIN {X 0,Y 759.906,Z 1256.49,A -85,B 0,C 180,E1 29058.769,E2 29058.769} C_VEL
LIN {X 0,Y 759.912,Z 1248.869,A -85,B 0,C 180,E1 29057.227,E2 29057.227} C_VEL
LIN {X 0,Y 759.914,Z 1240.113,A -85,B 0,C 180,E1 29055.677,E2 29055.677} C_VEL
LIN {X 0,Y 759.883,Z 1230.153,A -85,B 0,C 180,E1 29054.114,E2 29054.114} C_VEL
LIN {X 0,Y 759.89,Z 1217.147,A -85,B 0,C 180,E1 29052.302,E2 29052.302} C_VEL
LIN {X 0,Y 759.887,Z 1202.072,A -85,B 0,C 180,E1 29050.473,E2 29050.473} C_VEL
LIN {X 0,Y 759.903,Z 1188.815,A -85,B 0,C 180,E1 29049.027,E2 29049.027} C_VEL
LIN {X 0,Y 759.907,Z 1174.099,A -85,B 0,C 180,E1 29047.567,E2 29047.567} C_VEL
LIN {X 0,Y 759.891,Z 1155.368,A -85,B 0,C 180,E1 29045.884,E2 29045.884} C_VEL
LIN {X 0,Y 759.914,Z 1136.586,A -85,B 0,C 180,E1 29044.389,E2 29044.389} C_VEL
LIN {X 0,Y 759.918,Z 1119.359,A -85,B 0,C 180,E1 29043.139,E2 29043.139} C_VEL
LIN {X 0,Y 759.917,Z 1097.906,A -85,B 0,C 180,E1 29041.725,E2 29041.725} C_VEL
LIN {X 0,Y 759.907,Z 1075.541,A -85,B 0,C 180,E1 29040.43,E2 29040.43} C_VEL
LIN {X 0,Y 759.913,Z 1056.373,A -85,B 0,C 180,E1 29039.432,E2 29039.432} C_VEL
LIN {X 0,Y 759.912,Z 1037.641,A -85,B 0,C 180,E1 29038.552,E2 29038.552} C_VEL
LIN {X 0,Y 759.918,Z 1018.504,A -85,B 0,C 180,E1 29037.747,E2 29037.747} C_VEL
LIN {X 0,Y 759.919,Z 1000.794,A -85,B 0,C 180,E1 29037.083,E2 29037.083} C_VEL
LIN {X 0,Y 759.909,Z 982.458,A -85,B 0,C 180,E1 29036.472,E2 29036.472} C_VEL
LIN {X 0,Y 759.908,Z 960.584,A -85,B 0,C 180,E1 29035.837,E2 29035.837} C_VEL
LIN {X 0,Y 759.907,Z 932.692,A -85,B 0,C 180,E1 29035.192,E2 29035.192} C_VEL
LIN {X 0,Y 759.913,Z 905.983,A -85,B 0,C 180,E1 29034.735,E2 29034.735} C_VEL
LIN {X 0,Y 759.912,Z 800.731,A -85,B 0,C 180,E1 29033.51,E2 29033.51} C_VEL
LIN {X 0,Y 759.901,Z 583.545,A -85,B 0,C 180,E1 29030.965,E2 29030.965} C_VEL
LIN {X 0,Y 759.868,Z 427.536,A -85,B 0,C 180,E1 29029.069,E2 29029.069} C_VEL
LIN {X 0,Y 759.835,Z 396.582,A -85,B 0,C 180,E1 29027.026,E2 29027.026} C_VEL
LIN {X 0,Y 759.828,Z 396.578,A -85,B 0,C 180,E1 29023.96,E2 29023.96} C_VEL
LIN {X 0,Y 759.806,Z 396.577,A -85,B 0,C 180,E1 29021.549,E2 29021.549} C_VEL
LIN {X 0,Y 759.807,Z 396.577,A -85,B 0,C 180,E1 29019.368,E2 29019.368} C_VEL
LIN {X 0,Y 759.815,Z 396.576,A -85,B 0,C 180,E1 29017.111,E2 29017.111} C_VEL
LIN {X 0,Y 759.858,Z 396.577,A -85,B 0,C 180,E1 29014.643,E2 29014.643} C_VEL
LIN {X 0,Y 759.849,Z 396.573,A -85,B 0,C 180,E1 29011.637,E2 29011.637} C_VEL
LIN {X 0,Y 759.827,Z 396.574,A -85,B 0,C 180,E1 29009.224,E2 29009.224} C_VEL
LIN {X 0,Y 759.83,Z 396.575,A -85,B 0,C 180,E1 29006.916,E2 29006.916} C_VEL
LIN {X 0,Y 759.883,Z 396.576,A -85,B 0,C 180,E1 29004.322,E2 29004.322} C_VEL
LIN {X 0,Y 759.866,Z 396.57,A -85,B 0,C 180,E1 29001.377,E2 29001.377} C_VEL
LIN {X 0,Y 759.842,Z 396.572,A -85,B 0,C 180,E1 28998.888,E2 28998.888} C_VEL
LIN {X 0,Y 759.86,Z 396.575,A -85,B 0,C 180,E1 28996.409,E2 28996.409} C_VEL
LIN {X 0,Y 759.917,Z 396.567,A -85,B 0,C 180,E1 28993.468,E2 28993.468} C_VEL
LIN {X 0,Y 759.856,Z 396.57,A -85,B 0,C 180,E1 28990.769,E2 28990.769} C_VEL
LIN {X 0,Y 759.875,Z 396.573,A -85,B 0,C 180,E1 28988.17,E2 28988.17} C_VEL
LIN {X 0,Y 759.912,Z 396.566,A -85,B 0,C 180,E1 28985.209,E2 28985.209} C_VEL
LIN {X 0,Y 759.865,Z 396.569,A -85,B 0,C 180,E1 28982.489,E2 28982.489} C_VEL
LIN {X 0,Y 759.914,Z 396.578,A -85,B 0,C 180,E1 28979.698,E2 28979.698} C_VEL
LIN {X 0,Y 759.909,Z 396.565,A -85,B 0,C 180,E1 28977.059,E2 28977.059} C_VEL
LIN {X 0,Y 758.941,Z 396.686,A -85,B 0,C 180,E1 28976.478,E2 28976.478} C_VEL
LIN {X 0,Y 752.493,Z 397.489,A -85,B 0,C 180,E1 28974.852,E2 28974.852} C_VEL
LIN {X 0,Y 751.942,Z 397.557,A -85,B 0,C 180,E1 28974.429,E2 28974.429} C_VEL
LIN {X 0,Y 751.973,Z 397.564,A -85,B 0,C 180,E1 28971.589,E2 28971.589} C_VEL
LIN {X 0,Y 751.968,Z 397.553,A -85,B 0,C 180,E1 28968.515,E2 28968.515} C_VEL
LIN {X 0,Y 751.97,Z 397.564,A -85,B 0,C 180,E1 28965.523,E2 28965.523} C_VEL
LIN {X 0,Y 751.971,Z 397.553,A -85,B 0,C 180,E1 28962.512,E2 28962.512} C_VEL
LIN {X 0,Y 751.956,Z 397.561,A -85,B 0,C 180,E1 28959.611,E2 28959.611} C_VEL
LIN {X 0,Y 751.948,Z 397.56,A -85,B 0,C 180,E1 28956.821,E2 28956.821} C_VEL
LIN {X 0,Y 751.966,Z 397.552,A -85,B 0,C 180,E1 28953.972,E2 28953.972} C_VEL
LIN {X 0,Y 751.965,Z 397.563,A -85,B 0,C 180,E1 28951.038,E2 28951.038} C_VEL
LIN {X 0,Y 751.957,Z 397.555,A -85,B 0,C 180,E1 28948.136,E2 28948.136} C_VEL
LIN {X 0,Y 751.975,Z 397.563,A -85,B 0,C 180,E1 28945.126,E2 28945.126} C_VEL
LIN {X 0,Y 751.933,Z 397.557,A -85,B 0,C 180,E1 28942.288,E2 28942.288} C_VEL
LIN {X 0,Y 751.972,Z 397.557,A -85,B 0,C 180,E1 28939.516,E2 28939.516} C_VEL
LIN {X 0,Y 751.939,Z 397.565,A -85,B 0,C 180,E1 28936.569,E2 28936.569} C_VEL
LIN {X 0,Y 751.933,Z 397.561,A -85,B 0,C 180,E1 28933.853,E2 28933.853} C_VEL
LIN {X 0,Y 751.992,Z 397.756,A -85,B 0,C 180,E1 28932.75,E2 28932.75} C_VEL
LIN {X 0,Y 753.245,Z 401.563,A -85,B 0,C 180,E1 28932.403,E2 28932.403} C_VEL
LIN {X 0,Y 753.366,Z 418.371,A -85,B 0,C 180,E1 28931.296,E2 28931.296} C_VEL
LIN {X 0,Y 753.853,Z 421.381,A -85,B 0,C 180,E1 28931.226,E2 28931.226} C_VEL
LIN {X 0,Y 753.621,Z 634.289,A -85,B 0,C 180,E1 28928.647,E2 28928.647} C_VEL
LIN {X 0,Y 753.409,Z 859.235,A -85,B 0,C 180,E1 28926.017,E2 28926.017} C_VEL
LIN {X 0,Y 753.358,Z 899.26,A -85,B 0,C 180,E1 28925.525,E2 28925.525} C_VEL
LIN {X 0,Y 753.269,Z 925.507,A -85,B 0,C 180,E1 28925.055,E2 28925.055} C_VEL
LIN {X 0,Y 753.181,Z 952.198,A -85,B 0,C 180,E1 28924.423,E2 28924.423} C_VEL
LIN {X 0,Y 753.091,Z 978.285,A -85,B 0,C 180,E1 28923.645,E2 28923.645} C_VEL
LIN {X 0,Y 752.953,Z 1004.966,A -85,B 0,C 180,E1 28922.686,E2 28922.686} C_VEL
LIN {X 0,Y 752.859,Z 1025.653,A -85,B 0,C 180,E1 28921.822,E2 28921.822} C_VEL
LIN {X 0,Y 752.755,Z 1044.583,A -85,B 0,C 180,E1 28920.935,E2 28920.935} C_VEL
LIN {X 0,Y 752.664,Z 1063.976,A -85,B 0,C 180,E1 28919.924,E2 28919.924} C_VEL
LIN {X 0,Y 752.556,Z 1084.671,A -85,B 0,C 180,E1 28918.727,E2 28918.727} C_VEL
LIN {X 0,Y 752.425,Z 1107.966,A -85,B 0,C 180,E1 28917.204,E2 28917.204} C_VEL
LIN {X 0,Y 752.331,Z 1125.444,A -85,B 0,C 180,E1 28915.93,E2 28915.93} C_VEL
LIN {X 0,Y 752.261,Z 1143.299,A -85,B 0,C 180,E1 28914.502,E2 28914.502} C_VEL
LIN {X 0,Y 752.174,Z 1163.43,A -85,B 0,C 180,E1 28912.696,E2 28912.696} C_VEL
LIN {X 0,Y 752.104,Z 1178.387,A -85,B 0,C 180,E1 28911.2,E2 28911.2} C_VEL
LIN {X 0,Y 752.038,Z 1193.1,A -85,B 0,C 180,E1 28909.577,E2 28909.577} C_VEL
LIN {X 0,Y 751.973,Z 1209.216,A -85,B 0,C 180,E1 28907.562,E2 28907.562} C_VEL
LIN {X 0,Y 751.945,Z 1220.438,A -85,B 0,C 180,E1 28905.97,E2 28905.97} C_VEL
LIN {X 0,Y 751.958,Z 1230.314,A -85,B 0,C 180,E1 28904.4,E2 28904.4} C_VEL
LIN {X 0,Y 751.929,Z 1239.044,A -85,B 0,C 180,E1 28902.832,E2 28902.832} C_VEL
LIN {X 0,Y 751.924,Z 1246.998,A -85,B 0,C 180,E1 28901.197,E2 28901.197} C_VEL
LIN {X 0,Y 751.871,Z 1255,A -85,B 0,C 180,E1 28899.262,E2 28899.262} C_VEL
LIN {X 0,Y 751.915,Z 1262.216,A -85,B 0,C 180,E1 28897.029,E2 28897.029} C_VEL
LIN {X 0,Y 751.913,Z 1266.95,A -85,B 0,C 180,E1 28895.037,E2 28895.037} C_VEL
LIN {X 0,Y 751.909,Z 1270.227,A -85,B 0,C 180,E1 28892.975,E2 28892.975} C_VEL
LIN {X 0,Y 751.877,Z 1271.701,A -85,B 0,C 180,E1 28890.993,E2 28890.993} C_VEL
LIN {X 0,Y 751.864,Z 1271.841,A -85,B 0,C 180,E1 28889.393,E2 28889.393} C_VEL
LIN {X 0,Y 751.909,Z 1270.987,A -85,B 0,C 180,E1 28887.792,E2 28887.792} C_VEL
LIN {X 0,Y 751.915,Z 1268.88,A -85,B 0,C 180,E1 28885.961,E2 28885.961} C_VEL
LIN {X 0,Y 751.918,Z 1264.664,A -85,B 0,C 180,E1 28883.819,E2 28883.819} C_VEL
LIN {X 0,Y 751.913,Z 1258.973,A -85,B 0,C 180,E1 28881.822,E2 28881.822} C_VEL
LIN {X 0,Y 751.908,Z 1252.925,A -85,B 0,C 180,E1 28880.125,E2 28880.125} C_VEL
LIN {X 0,Y 751.929,Z 1246.003,A -85,B 0,C 180,E1 28878.497,E2 28878.497} C_VEL
LIN {X 0,Y 751.916,Z 1238.309,A -85,B 0,C 180,E1 28876.937,E2 28876.937} C_VEL
LIN {X 0,Y 751.948,Z 1229.011,A -85,B 0,C 180,E1 28875.29,E2 28875.29} C_VEL
LIN {X 0,Y 752.002,Z 1216.253,A -85,B 0,C 180,E1 28873.313,E2 28873.313} C_VEL
LIN {X 0,Y 752.033,Z 1202.199,A -85,B 0,C 180,E1 28871.441,E2 28871.441} C_VEL
LIN {X 0,Y 752.042,Z 1189.667,A -85,B 0,C 180,E1 28869.942,E2 28869.942} C_VEL
LIN {X 0,Y 752.118,Z 1175.39,A -85,B 0,C 180,E1 28868.396,E2 28868.396} C_VEL
LIN {X 0,Y 752.203,Z 1155.781,A -85,B 0,C 180,E1 28866.501,E2 28866.501} C_VEL
LIN {X 0,Y 752.285,Z 1139.37,A -85,B 0,C 180,E1 28865.085,E2 28865.085} C_VEL
LIN {X 0,Y 752.339,Z 1121.146,A -85,B 0,C 180,E1 28863.651,E2 28863.651} C_VEL
LIN {X 0,Y 752.476,Z 1098.823,A -85,B 0,C 180,E1 28862.087,E2 28862.087} C_VEL
LIN {X 0,Y 752.58,Z 1080.055,A -85,B 0,C 180,E1 28860.908,E2 28860.908} C_VEL
LIN {X 0,Y 752.67,Z 1061.699,A -85,B 0,C 180,E1 28859.861,E2 28859.861} C_VEL
LIN {X 0,Y 752.771,Z 1041.149,A -85,B 0,C 180,E1 28858.804,E2 28858.804} C_VEL
LIN {X 0,Y 752.932,Z 1014.498,A -85,B 0,C 180,E1 28857.608,E2 28857.608} C_VEL
LIN {X 0,Y 753.025,Z 993.009,A -85,B 0,C 180,E1 28856.776,E2 28856.776} C_VEL
LIN {X 0,Y 753.102,Z 973.39,A -85,B 0,C 180,E1 28856.112,E2 28856.112} C_VEL
LIN {X 0,Y 753.193,Z 950.466,A -85,B 0,C 180,E1 28855.441,E2 28855.441} C_VEL
LIN {X 0,Y 753.279,Z 922.904,A -85,B 0,C 180,E1 28854.8,E2 28854.8} C_VEL
LIN {X 0,Y 753.355,Z 895.487,A -85,B 0,C 180,E1 28854.33,E2 28854.33} C_VEL
LIN {X 0,Y 753.602,Z 649.163,A -85,B 0,C 180,E1 28851.439,E2 28851.439} C_VEL
LIN {X 0,Y 753.806,Z 442.4,A -85,B 0,C 180,E1 28848.941,E2 28848.941} C_VEL
LIN {X 0,Y 753.68,Z 419.539,A -85,B 0,C 180,E1 28848.649,E2 28848.649} C_VEL
LIN {X 0,Y 753.237,Z 417.742,A -85,B 0,C 180,E1 28848.592,E2 28848.592} C_VEL
LIN {X 0,Y 753.168,Z 400.96,A -85,B 0,C 180,E1 28847.46,E2 28847.46} C_VEL
LIN {X 0,Y 751.96,Z 397.568,A -85,B 0,C 180,E1 28847.126,E2 28847.126} C_VEL
LIN {X 0,Y 751.927,Z 397.56,A -85,B 0,C 180,E1 28844.11,E2 28844.11} C_VEL
LIN {X 0,Y 751.905,Z 397.561,A -85,B 0,C 180,E1 28841.573,E2 28841.573} C_VEL
LIN {X 0,Y 751.929,Z 397.565,A -85,B 0,C 180,E1 28839.058,E2 28839.058} C_VEL
LIN {X 0,Y 751.946,Z 397.558,A -85,B 0,C 180,E1 28835.997,E2 28835.997} C_VEL
LIN {X 0,Y 751.902,Z 397.56,A -85,B 0,C 180,E1 28833.38,E2 28833.38} C_VEL
LIN {X 0,Y 751.915,Z 397.564,A -85,B 0,C 180,E1 28830.884,E2 28830.884} C_VEL
LIN {X 0,Y 751.978,Z 397.559,A -85,B 0,C 180,E1 28827.994,E2 28827.994} C_VEL
LIN {X 0,Y 751.906,Z 397.558,A -85,B 0,C 180,E1 28825.269,E2 28825.269} C_VEL
LIN {X 0,Y 751.898,Z 397.563,A -85,B 0,C 180,E1 28822.849,E2 28822.849} C_VEL
LIN {X 0,Y 751.932,Z 397.564,A -85,B 0,C 180,E1 28820.308,E2 28820.308} C_VEL
LIN {X 0,Y 751.926,Z 397.56,A -85,B 0,C 180,E1 28817.25,E2 28817.25} C_VEL
LIN {X 0,Y 751.894,Z 397.559,A -85,B 0,C 180,E1 28814.793,E2 28814.793} C_VEL
LIN {X 0,Y 751.895,Z 397.563,A -85,B 0,C 180,E1 28812.441,E2 28812.441} C_VEL
LIN {X 0,Y 751.938,Z 397.565,A -85,B 0,C 180,E1 28809.85,E2 28809.85} C_VEL
LIN {X 0,Y 751.921,Z 397.56,A -85,B 0,C 180,E1 28806.874,E2 28806.874} C_VEL
LIN {X 0,Y 751.891,Z 397.562,A -85,B 0,C 180,E1 28804.424,E2 28804.424} C_VEL
LIN {X 0,Y 751.891,Z 397.561,A -85,B 0,C 180,E1 28802.058,E2 28802.058} C_VEL
LIN {X 0,Y 751.938,Z 397.566,A -85,B 0,C 180,E1 28799.467,E2 28799.467} C_VEL
LIN {X 0,Y 751.915,Z 397.559,A -85,B 0,C 180,E1 28796.493,E2 28796.493} C_VEL
LIN {X 0,Y 751.887,Z 397.563,A -85,B 0,C 180,E1 28794.046,E2 28794.046} C_VEL
LIN {X 0,Y 751.885,Z 397.563,A -85,B 0,C 180,E1 28791.742,E2 28791.742} C_VEL
LIN {X 0,Y 751.906,Z 397.563,A -85,B 0,C 180,E1 28789.308,E2 28789.308} C_VEL
LIN {X 0,Y 751.935,Z 397.56,A -85,B 0,C 180,E1 28786.308,E2 28786.308} C_VEL
LIN {X 0,Y 751.885,Z 397.562,A -85,B 0,C 180,E1 28783.752,E2 28783.752} C_VEL
LIN {X 0,Y 751.879,Z 397.564,A -85,B 0,C 180,E1 28781.46,E2 28781.46} C_VEL
LIN {X 0,Y 751.883,Z 397.561,A -85,B 0,C 180,E1 28779.196,E2 28779.196} C_VEL
LIN {X 0,Y 751.945,Z 397.566,A -85,B 0,C 180,E1 28776.554,E2 28776.554} C_VEL
LIN {X 0,Y 751.899,Z 397.563,A -85,B 0,C 180,E1 28773.63,E2 28773.63} C_VEL
LIN {X 0,Y 751.878,Z 397.564,A -85,B 0,C 180,E1 28771.309,E2 28771.309} C_VEL
LIN {X 0,Y 751.874,Z 397.564,A -85,B 0,C 180,E1 28769.114,E2 28769.114} C_VEL
LIN {X 0,Y 751.873,Z 397.565,A -85,B 0,C 180,E1 28766.867,E2 28766.867} C_VEL
LIN {X 0,Y 751.88,Z 397.565,A -85,B 0,C 180,E1 28764.599,E2 28764.599} C_VEL
LIN {X 0,Y 751.977,Z 397.566,A -85,B 0,C 180,E1 28761.791,E2 28761.791} C_VEL
LIN {X 0,Y 751.883,Z 397.563,A -85,B 0,C 180,E1 28759.033,E2 28759.033} C_VEL
LIN {X 0,Y 751.871,Z 397.567,A -85,B 0,C 180,E1 28756.773,E2 28756.773} C_VEL
LIN {X 0,Y 751.867,Z 397.569,A -85,B 0,C 180,E1 28754.596,E2 28754.596} C_VEL
LIN {X 0,Y 751.991,Z 397.696,A -85,B 0,C 180,E1 28753.433,E2 28753.433} C_VEL
LIN {X 0,Y 753.262,Z 401.68,A -85,B 0,C 180,E1 28753.074,E2 28753.074} C_VEL
LIN {X 0,Y 753.34,Z 428.194,A -85,B 0,C 180,E1 28751.345,E2 28751.345} C_VEL
LIN {X 0,Y 753.801,Z 431.232,A -85,B 0,C 180,E1 28751.277,E2 28751.277} C_VEL
LIN {X 0,Y 753.639,Z 629.182,A -85,B 0,C 180,E1 28748.872,E2 28748.872} C_VEL
LIN {X 0,Y 753.421,Z 850.699,A -85,B 0,C 180,E1 28746.275,E2 28746.275} C_VEL
LIN {X 0,Y 753.355,Z 907.13,A -85,B 0,C 180,E1 28745.601,E2 28745.601} C_VEL
LIN {X 0,Y 753.272,Z 933.851,A -85,B 0,C 180,E1 28745.135,E2 28745.135} C_VEL
LIN {X 0,Y 753.187,Z 961.205,A -85,B 0,C 180,E1 28744.494,E2 28744.494} C_VEL
LIN {X 0,Y 753.098,Z 984.882,A -85,B 0,C 180,E1 28743.796,E2 28743.796} C_VEL
LIN {X 0,Y 752.994,Z 1010.299,A -85,B 0,C 180,E1 28742.917,E2 28742.917} C_VEL
LIN {X 0,Y 752.858,Z 1034.778,A -85,B 0,C 180,E1 28741.906,E2 28741.906} C_VEL
LIN {X 0,Y 752.756,Z 1054.699,A -85,B 0,C 180,E1 28740.974,E2 28740.974} C_VEL
LIN {X 0,Y 752.662,Z 1074.089,A -85,B 0,C 180,E1 28739.963,E2 28739.963} C_VEL
LIN {X 0,Y 752.557,Z 1095.423,A -85,B 0,C 180,E1 28738.727,E2 28738.727} C_VEL
LIN {X 0,Y 752.424,Z 1117.976,A -85,B 0,C 180,E1 28737.248,E2 28737.248} C_VEL
LIN {X 0,Y 752.332,Z 1135.543,A -85,B 0,C 180,E1 28735.968,E2 28735.968} C_VEL
LIN {X 0,Y 752.26,Z 1153.396,A -85,B 0,C 180,E1 28734.539,E2 28734.539} C_VEL
LIN {X 0,Y 752.174,Z 1173.297,A -85,B 0,C 180,E1 28732.754,E2 28732.754} C_VEL
LIN {X 0,Y 752.105,Z 1188.262,A -85,B 0,C 180,E1 28731.259,E2 28731.259} C_VEL
LIN {X 0,Y 752.036,Z 1202.229,A -85,B 0,C 180,E1 28729.721,E2 28729.721} C_VEL
LIN {X 0,Y 751.991,Z 1217.775,A -85,B 0,C 180,E1 28727.804,E2 28727.804} C_VEL
LIN {X 0,Y 751.949,Z 1230.185,A -85,B 0,C 180,E1 28726.053,E2 28726.053} C_VEL
LIN {X 0,Y 751.961,Z 1240.141,A -85,B 0,C 180,E1 28724.474,E2 28724.474} C_VEL
LIN {X 0,Y 751.928,Z 1248.893,A -85,B 0,C 180,E1 28722.906,E2 28722.906} C_VEL
LIN {X 0,Y 751.928,Z 1256.511,A -85,B 0,C 180,E1 28721.347,E2 28721.347} C_VEL
LIN {X 0,Y 751.888,Z 1263.665,A -85,B 0,C 180,E1 28719.643,E2 28719.643} C_VEL
LIN {X 0,Y 751.89,Z 1271.04,A -85,B 0,C 180,E1 28717.486,E2 28717.486} C_VEL
LIN {X 0,Y 751.907,Z 1276.285,A -85,B 0,C 180,E1 28715.415,E2 28715.415} C_VEL
LIN {X 0,Y 751.908,Z 1279.792,A -85,B 0,C 180,E1 28713.352,E2 28713.352} C_VEL
LIN {X 0,Y 751.884,Z 1281.671,A -85,B 0,C 180,E1 28711.141,E2 28711.141} C_VEL
LIN {X 0,Y 751.865,Z 1281.849,A -85,B 0,C 180,E1 28709.464,E2 28709.464} C_VEL
LIN {X 0,Y 751.913,Z 1281.011,A -85,B 0,C 180,E1 28707.864,E2 28707.864} C_VEL
LIN {X 0,Y 751.912,Z 1278.925,A -85,B 0,C 180,E1 28706.033,E2 28706.033} C_VEL
LIN {X 0,Y 751.917,Z 1274.73,A -85,B 0,C 180,E1 28703.891,E2 28703.891} C_VEL
LIN {X 0,Y 751.898,Z 1269.321,A -85,B 0,C 180,E1 28701.972,E2 28701.972} C_VEL
LIN {X 0,Y 751.906,Z 1263.023,A -85,B 0,C 180,E1 28700.195,E2 28700.195} C_VEL
LIN {X 0,Y 751.927,Z 1256.133,A -85,B 0,C 180,E1 28698.57,E2 28698.57} C_VEL
LIN {X 0,Y 751.919,Z 1248.459,A -85,B 0,C 180,E1 28697.011,E2 28697.011} C_VEL
LIN {X 0,Y 751.959,Z 1239.649,A -85,B 0,C 180,E1 28695.443,E2 28695.443} C_VEL
LIN {X 0,Y 751.959,Z 1228.587,A -85,B 0,C 180,E1 28693.704,E2 28693.704} C_VEL
LIN {X 0,Y 752.025,Z 1213.362,A -85,B 0,C 180,E1 28691.631,E2 28691.631} C_VEL
LIN {X 0,Y 752.04,Z 1200.252,A -85,B 0,C 180,E1 28690.054,E2 28690.054} C_VEL
LIN {X 0,Y 752.116,Z 1186.477,A -85,B 0,C 180,E1 28688.555,E2 28688.555} C_VEL
LIN {X 0,Y 752.194,Z 1168.481,A -85,B 0,C 180,E1 28686.787,E2 28686.787} C_VEL
LIN {X 0,Y 752.281,Z 1150.277,A -85,B 0,C 180,E1 28685.205,E2 28685.205} C_VEL
LIN {X 0,Y 752.333,Z 1133.264,A -85,B 0,C 180,E1 28683.858,E2 28683.858} C_VEL
LIN {X 0,Y 752.477,Z 1111.16,A -85,B 0,C 180,E1 28682.284,E2 28682.284} C_VEL
LIN {X 0,Y 752.573,Z 1090.674,A -85,B 0,C 180,E1 28680.99,E2 28680.99} C_VEL
LIN {X 0,Y 752.668,Z 1072.39,A -85,B 0,C 180,E1 28679.944,E2 28679.944} C_VEL
LIN {X 0,Y 752.762,Z 1052.816,A -85,B 0,C 180,E1 28678.932,E2 28678.932} C_VEL
LIN {X 0,Y 752.91,Z 1028.68,A -85,B 0,C 180,E1 28677.822,E2 28677.822} C_VEL
LIN {X 0,Y 753.022,Z 1004.614,A -85,B 0,C 180,E1 28676.879,E2 28676.879} C_VEL
LIN {X 0,Y 753.1,Z 983.98,A -85,B 0,C 180,E1 28676.176,E2 28676.176} C_VEL
LIN {X 0,Y 753.191,Z 960.747,A -85,B 0,C 180,E1 28675.494,E2 28675.494} C_VEL
LIN {X 0,Y 753.277,Z 933.105,A -85,B 0,C 180,E1 28674.849,E2 28674.849} C_VEL
LIN {X 0,Y 753.355,Z 905.973,A -85,B 0,C 180,E1 28674.382,E2 28674.382} C_VEL
LIN {X 0,Y 753.604,Z 657.723,A -85,B 0,C 180,E1 28671.467,E2 28671.467} C_VEL
LIN {X 0,Y 753.767,Z 459.236,A -85,B 0,C 180,E1 28669.068,E2 28669.068} C_VEL
LIN {X 0,Y 753.633,Z 429.334,A -85,B 0,C 180,E1 28668.689,E2 28668.689} C_VEL
LIN {X 0,Y 753.229,Z 427.342,A -85,B 0,C 180,E1 28668.617,E2 28668.617} C_VEL
LIN {X 0,Y 753.116,Z 400.89,A -85,B 0,C 180,E1 28666.862,E2 28666.862} C_VEL
LIN {X 0,Y 751.974,Z 397.566,A -85,B 0,C 180,E1 28666.553,E2 28666.553} C_VEL
LIN {X 0,Y 751.871,Z 397.569,A -85,B 0,C 180,E1 28663.752,E2 28663.752} C_VEL
LIN {X 0,Y 751.866,Z 397.565,A -85,B 0,C 180,E1 28661.405,E2 28661.405} C_VEL
LIN {X 0,Y 751.87,Z 397.567,A -85,B 0,C 180,E1 28659.273,E2 28659.273} C_VEL
LIN {X 0,Y 751.888,Z 397.564,A -85,B 0,C 180,E1 28656.943,E2 28656.943} C_VEL
LIN {X 0,Y 751.961,Z 397.562,A -85,B 0,C 180,E1 28654.043,E2 28654.043} C_VEL
LIN {X 0,Y 751.889,Z 397.563,A -85,B 0,C 180,E1 28651.378,E2 28651.378} C_VEL
LIN {X 0,Y 751.888,Z 397.563,A -85,B 0,C 180,E1 28649.038,E2 28649.038} C_VEL
LIN {X 0,Y 751.91,Z 397.565,A -85,B 0,C 180,E1 28646.625,E2 28646.625} C_VEL
LIN {X 0,Y 751.951,Z 397.56,A -85,B 0,C 180,E1 28643.627,E2 28643.627} C_VEL
LIN {X 0,Y 751.901,Z 397.56,A -85,B 0,C 180,E1 28641.009,E2 28641.009} C_VEL
LIN {X 0,Y 751.913,Z 397.563,A -85,B 0,C 180,E1 28638.531,E2 28638.531} C_VEL
LIN {X 0,Y 751.975,Z 397.557,A -85,B 0,C 180,E1 28635.702,E2 28635.702} C_VEL
LIN {X 0,Y 751.919,Z 397.559,A -85,B 0,C 180,E1 28632.909,E2 28632.909} C_VEL
LIN {X 0,Y 751.924,Z 397.563,A -85,B 0,C 180,E1 28630.342,E2 28630.342} C_VEL
LIN {X 0,Y 751.972,Z 397.559,A -85,B 0,C 180,E1 28627.488,E2 28627.488} C_VEL
LIN {X 0,Y 751.931,Z 397.557,A -85,B 0,C 180,E1 28624.729,E2 28624.729} C_VEL
LIN {X 0,Y 751.947,Z 397.561,A -85,B 0,C 180,E1 28621.981,E2 28621.981} C_VEL
LIN {X 0,Y 751.976,Z 397.553,A -85,B 0,C 180,E1 28619.01,E2 28619.01} C_VEL
LIN {X 0,Y 751.934,Z 397.557,A -85,B 0,C 180,E1 28616.188,E2 28616.188} C_VEL
LIN {X 0,Y 751.942,Z 397.557,A -85,B 0,C 180,E1 28614.429,E2 28614.429} C_VEL
LIN {X 0,Y 750.93,Z 397.692,A -85,B 0,C 180,E1 28613.842,E2 28613.842} C_VEL
LIN {X 0,Y 744.52,Z 398.483,A -85,B 0,C 180,E1 28612.198,E2 28612.198} C_VEL
LIN {X 0,Y 744.016,Z 398.552,A -85,B 0,C 180,E1 28611.771,E2 28611.771} C_VEL
LIN {X 0,Y 744.027,Z 398.544,A -85,B 0,C 180,E1 28608.822,E2 28608.822} C_VEL
LIN {X 0,Y 744.007,Z 398.547,A -85,B 0,C 180,E1 28606.001,E2 28606.001} C_VEL
LIN {X 0,Y 744.026,Z 398.553,A -85,B 0,C 180,E1 28603.206,E2 28603.206} C_VEL
LIN {X 0,Y 744.036,Z 398.539,A -85,B 0,C 180,E1 28600.287,E2 28600.287} C_VEL
LIN {X 0,Y 744.032,Z 398.555,A -85,B 0,C 180,E1 28597.23,E2 28597.23} C_VEL
LIN {X 0,Y 744.03,Z 398.538,A -85,B 0,C 180,E1 28594.188,E2 28594.188} C_VEL
LIN {X 0,Y 744.031,Z 398.553,A -85,B 0,C 180,E1 28591.154,E2 28591.154} C_VEL
LIN {X 0,Y 744.008,Z 398.546,A -85,B 0,C 180,E1 28588.288,E2 28588.288} C_VEL
LIN {X 0,Y 744.024,Z 398.546,A -85,B 0,C 180,E1 28585.45,E2 28585.45} C_VEL
LIN {X 0,Y 743.999,Z 398.548,A -85,B 0,C 180,E1 28582.594,E2 28582.594} C_VEL
LIN {X 0,Y 744.018,Z 398.546,A -85,B 0,C 180,E1 28579.828,E2 28579.828} C_VEL
LIN {X 0,Y 744.016,Z 398.557,A -85,B 0,C 180,E1 28576.733,E2 28576.733} C_VEL
LIN {X 0,Y 743.986,Z 398.554,A -85,B 0,C 180,E1 28574.014,E2 28574.014} C_VEL
LIN {X 0,Y 744.057,Z 398.727,A -85,B 0,C 180,E1 28573.251,E2 28573.251} C_VEL
LIN {X 0,Y 745.43,Z 402.174,A -85,B 0,C 180,E1 28572.913,E2 28572.913} C_VEL
LIN {X 0,Y 746.631,Z 405.238,A -85,B 0,C 180,E1 28572.617,E2 28572.617} C_VEL
LIN {X 0,Y 746.724,Z 418.353,A -85,B 0,C 180,E1 28571.746,E2 28571.746} C_VEL
LIN {X 0,Y 747.823,Z 423.141,A -85,B 0,C 180,E1 28571.611,E2 28571.611} C_VEL
LIN {X 0,Y 747.362,Z 636.197,A -85,B 0,C 180,E1 28569.01,E2 28569.01} C_VEL
LIN {X 0,Y 746.927,Z 861.194,A -85,B 0,C 180,E1 28566.357,E2 28566.357} C_VEL
LIN {X 0,Y 746.824,Z 900.211,A -85,B 0,C 180,E1 28565.87,E2 28565.87} C_VEL
LIN {X 0,Y 746.657,Z 926.583,A -85,B 0,C 180,E1 28565.389,E2 28565.389} C_VEL
LIN {X 0,Y 746.482,Z 952.963,A -85,B 0,C 180,E1 28564.756,E2 28564.756} C_VEL
LIN {X 0,Y 746.288,Z 980.607,A -85,B 0,C 180,E1 28563.921,E2 28563.921} C_VEL
LIN {X 0,Y 746.013,Z 1005.339,A -85,B 0,C 180,E1 28563.014,E2 28563.014} C_VEL
LIN {X 0,Y 745.816,Z 1026.762,A -85,B 0,C 180,E1 28562.108,E2 28562.108} C_VEL
LIN {X 0,Y 745.613,Z 1046.377,A -85,B 0,C 180,E1 28561.175,E2 28561.175} C_VEL
LIN {X 0,Y 745.417,Z 1067.198,A -85,B 0,C 180,E1 28560.068,E2 28560.068} C_VEL
LIN {X 0,Y 745.117,Z 1091.871,A -85,B 0,C 180,E1 28558.582,E2 28558.582} C_VEL
LIN {X 0,Y 744.94,Z 1110.683,A -85,B 0,C 180,E1 28557.306,E2 28557.306} C_VEL
LIN {X 0,Y 744.768,Z 1129.432,A -85,B 0,C 180,E1 28555.906,E2 28555.906} C_VEL
LIN {X 0,Y 744.525,Z 1150.068,A -85,B 0,C 180,E1 28554.182,E2 28554.182} C_VEL
LIN {X 0,Y 744.43,Z 1165.349,A -85,B 0,C 180,E1 28552.759,E2 28552.759} C_VEL
LIN {X 0,Y 744.306,Z 1179.953,A -85,B 0,C 180,E1 28551.268,E2 28551.268} C_VEL
LIN {X 0,Y 744.189,Z 1196.561,A -85,B 0,C 180,E1 28549.384,E2 28549.384} C_VEL
LIN {X 0,Y 744.067,Z 1210.331,A -85,B 0,C 180,E1 28547.601,E2 28547.601} C_VEL
LIN {X 0,Y 744.012,Z 1220.908,A -85,B 0,C 180,E1 28546.074,E2 28546.074} C_VEL
LIN {X 0,Y 744.008,Z 1230.318,A -85,B 0,C 180,E1 28544.557,E2 28544.557} C_VEL
LIN {X 0,Y 743.948,Z 1239.048,A -85,B 0,C 180,E1 28542.972,E2 28542.972} C_VEL
LIN {X 0,Y 743.948,Z 1247.002,A -85,B 0,C 180,E1 28541.318,E2 28541.318} C_VEL
LIN {X 0,Y 743.882,Z 1255.002,A -85,B 0,C 180,E1 28539.362,E2 28539.362} C_VEL
LIN {X 0,Y 743.921,Z 1262.218,A -85,B 0,C 180,E1 28537.105,E2 28537.105} C_VEL
LIN {X 0,Y 743.911,Z 1266.951,A -85,B 0,C 180,E1 28535.091,E2 28535.091} C_VEL
LIN {X 0,Y 743.908,Z 1270.228,A -85,B 0,C 180,E1 28533.007,E2 28533.007} C_VEL
LIN {X 0,Y 743.878,Z 1271.701,A -85,B 0,C 180,E1 28531.003,E2 28531.003} C_VEL
LIN {X 0,Y 743.864,Z 1271.841,A -85,B 0,C 180,E1 28529.386,E2 28529.386} C_VEL
LIN {X 0,Y 743.908,Z 1270.987,A -85,B 0,C 180,E1 28527.768,E2 28527.768} C_VEL
LIN {X 0,Y 743.917,Z 1268.88,A -85,B 0,C 180,E1 28525.917,E2 28525.917} C_VEL
LIN {X 0,Y 743.921,Z 1264.663,A -85,B 0,C 180,E1 28523.752,E2 28523.752} C_VEL
LIN {X 0,Y 743.926,Z 1258.972,A -85,B 0,C 180,E1 28521.734,E2 28521.734} C_VEL
LIN {X 0,Y 743.929,Z 1252.924,A -85,B 0,C 180,E1 28520.018,E2 28520.018} C_VEL
LIN {X 0,Y 743.938,Z 1246.002,A -85,B 0,C 180,E1 28518.372,E2 28518.372} C_VEL
LIN {X 0,Y 743.938,Z 1238.307,A -85,B 0,C 180,E1 28516.795,E2 28516.795} C_VEL
LIN {X 0,Y 743.989,Z 1229.009,A -85,B 0,C 180,E1 28515.129,E2 28515.129} C_VEL
LIN {X 0,Y 744.082,Z 1216.247,A -85,B 0,C 180,E1 28513.13,E2 28513.13} C_VEL
LIN {X 0,Y 744.159,Z 1202.468,A -85,B 0,C 180,E1 28511.272,E2 28511.272} C_VEL
LIN {X 0,Y 744.221,Z 1189.341,A -85,B 0,C 180,E1 28509.685,E2 28509.685} C_VEL
LIN {X 0,Y 744.327,Z 1174.607,A -85,B 0,C 180,E1 28508.075,E2 28508.075} C_VEL
LIN {X 0,Y 744.524,Z 1155.31,A -85,B 0,C 180,E1 28506.202,E2 28506.202} C_VEL
LIN {X 0,Y 744.655,Z 1138.872,A -85,B 0,C 180,E1 28504.771,E2 28504.771} C_VEL
LIN {X 0,Y 744.885,Z 1118.921,A -85,B 0,C 180,E1 28503.194,E2 28503.194} C_VEL
LIN {X 0,Y 745.074,Z 1097.309,A -85,B 0,C 180,E1 28501.685,E2 28501.685} C_VEL
LIN {X 0,Y 745.275,Z 1078.592,A -85,B 0,C 180,E1 28500.507,E2 28500.507} C_VEL
LIN {X 0,Y 745.474,Z 1057.675,A -85,B 0,C 180,E1 28499.317,E2 28499.317} C_VEL
LIN {X 0,Y 745.784,Z 1031.731,A -85,B 0,C 180,E1 28498.027,E2 28498.027} C_VEL
LIN {X 0,Y 745.986,Z 1011.02,A -85,B 0,C 180,E1 28497.127,E2 28497.127} C_VEL
LIN {X 0,Y 746.169,Z 990.916,A -85,B 0,C 180,E1 28496.356,E2 28496.356} C_VEL
LIN {X 0,Y 746.335,Z 971.176,A -85,B 0,C 180,E1 28495.693,E2 28495.693} C_VEL
LIN {X 0,Y 746.517,Z 948.879,A -85,B 0,C 180,E1 28495.047,E2 28495.047} C_VEL
LIN {X 0,Y 746.702,Z 922.046,A -85,B 0,C 180,E1 28494.426,E2 28494.426} C_VEL
LIN {X 0,Y 746.836,Z 893.852,A -85,B 0,C 180,E1 28493.946,E2 28493.946} C_VEL
LIN {X 0,Y 747.323,Z 652.677,A -85,B 0,C 180,E1 28491.097,E2 28491.097} C_VEL
LIN {X 0,Y 747.742,Z 446.751,A -85,B 0,C 180,E1 28488.59,E2 28488.59} C_VEL
LIN {X 0,Y 747.644,Z 421.642,A -85,B 0,C 180,E1 28488.268,E2 28488.268} C_VEL
LIN {X 0,Y 746.601,Z 417.528,A -85,B 0,C 180,E1 28488.127,E2 28488.127} C_VEL
LIN {X 0,Y 746.546,Z 405.091,A -85,B 0,C 180,E1 28487.277,E2 28487.277} C_VEL
LIN {X 0,Y 744.039,Z 398.552,A -85,B 0,C 180,E1 28486.635,E2 28486.635} C_VEL
LIN {X 0,Y 743.973,Z 398.552,A -85,B 0,C 180,E1 28483.908,E2 28483.908} C_VEL
LIN {X 0,Y 743.971,Z 398.551,A -85,B 0,C 180,E1 28481.395,E2 28481.395} C_VEL
LIN {X 0,Y 744.038,Z 398.554,A -85,B 0,C 180,E1 28478.674,E2 28478.674} C_VEL
LIN {X 0,Y 743.978,Z 398.549,A -85,B 0,C 180,E1 28475.739,E2 28475.739} C_VEL
LIN {X 0,Y 743.963,Z 398.55,A -85,B 0,C 180,E1 28473.254,E2 28473.254} C_VEL
LIN {X 0,Y 744.005,Z 398.554,A -85,B 0,C 180,E1 28470.621,E2 28470.621} C_VEL
LIN {X 0,Y 743.991,Z 398.548,A -85,B 0,C 180,E1 28467.624,E2 28467.624} C_VEL
LIN {X 0,Y 743.959,Z 398.547,A -85,B 0,C 180,E1 28465.047,E2 28465.047} C_VEL
LIN {X 0,Y 743.972,Z 398.553,A -85,B 0,C 180,E1 28462.596,E2 28462.596} C_VEL
LIN {X 0,Y 744.039,Z 398.547,A -85,B 0,C 180,E1 28459.713,E2 28459.713} C_VEL
LIN {X 0,Y 743.962,Z 398.55,A -85,B 0,C 180,E1 28456.957,E2 28456.957} C_VEL
LIN {X 0,Y 743.954,Z 398.547,A -85,B 0,C 180,E1 28454.556,E2 28454.556} C_VEL
LIN {X 0,Y 743.989,Z 398.554,A -85,B 0,C 180,E1 28452.024,E2 28452.024} C_VEL
LIN {X 0,Y 743.985,Z 398.545,A -85,B 0,C 180,E1 28448.969,E2 28448.969} C_VEL
LIN {X 0,Y 743.954,Z 398.551,A -85,B 0,C 180,E1 28446.482,E2 28446.482} C_VEL
LIN {X 0,Y 743.955,Z 398.552,A -85,B 0,C 180,E1 28444.085,E2 28444.085} C_VEL
LIN {X 0,Y 744.026,Z 398.551,A -85,B 0,C 180,E1 28441.386,E2 28441.386} C_VEL
LIN {X 0,Y 743.966,Z 398.549,A -85,B 0,C 180,E1 28438.46,E2 28438.46} C_VEL
LIN {X 0,Y 743.947,Z 398.548,A -85,B 0,C 180,E1 28436.07,E2 28436.07} C_VEL
LIN {X 0,Y 743.949,Z 398.553,A -85,B 0,C 180,E1 28433.75,E2 28433.75} C_VEL
LIN {X 0,Y 743.993,Z 398.553,A -85,B 0,C 180,E1 28431.187,E2 28431.187} C_VEL
LIN {X 0,Y 743.974,Z 398.551,A -85,B 0,C 180,E1 28428.212,E2 28428.212} C_VEL
LIN {X 0,Y 743.944,Z 398.55,A -85,B 0,C 180,E1 28425.761,E2 28425.761} C_VEL
LIN {X 0,Y 743.941,Z 398.551,A -85,B 0,C 180,E1 28423.525,E2 28423.525} C_VEL
LIN {X 0,Y 743.95,Z 398.554,A -85,B 0,C 180,E1 28421.182,E2 28421.182} C_VEL
LIN {X 0,Y 744.039,Z 398.552,A -85,B 0,C 180,E1 28418.394,E2 28418.394} C_VEL
LIN {X 0,Y 743.953,Z 398.551,A -85,B 0,C 180,E1 28415.631,E2 28415.631} C_VEL
LIN {X 0,Y 743.937,Z 398.553,A -85,B 0,C 180,E1 28413.24,E2 28413.24} C_VEL
LIN {X 0,Y 743.935,Z 398.553,A -85,B 0,C 180,E1 28411.033,E2 28411.033} C_VEL
LIN {X 0,Y 743.945,Z 398.553,A -85,B 0,C 180,E1 28408.73,E2 28408.73} C_VEL
LIN {X 0,Y 744.039,Z 398.55,A -85,B 0,C 180,E1 28405.868,E2 28405.868} C_VEL
LIN {X 0,Y 743.941,Z 398.554,A -85,B 0,C 180,E1 28403.095,E2 28403.095} C_VEL
LIN {X 0,Y 743.931,Z 398.556,A -85,B 0,C 180,E1 28400.823,E2 28400.823} C_VEL
LIN {X 0,Y 743.931,Z 398.552,A -85,B 0,C 180,E1 28398.583,E2 28398.583} C_VEL
LIN {X 0,Y 743.939,Z 398.558,A -85,B 0,C 180,E1 28396.303,E2 28396.303} C_VEL
LIN {X 0,Y 743.981,Z 398.693,A -85,B 0,C 180,E1 28393.951,E2 28393.951} C_VEL
LIN {X 0,Y 745.067,Z 401.654,A -85,B 0,C 180,E1 28393.668,E2 28393.668} C_VEL
LIN {X 0,Y 746.704,Z 405.336,A -85,B 0,C 180,E1 28393.299,E2 28393.299} C_VEL
LIN {X 0,Y 746.734,Z 428.165,A -85,B 0,C 180,E1 28391.793,E2 28391.793} C_VEL
LIN {X 0,Y 747.77,Z 432.924,A -85,B 0,C 180,E1 28391.662,E2 28391.662} C_VEL
LIN {X 0,Y 747.395,Z 631.112,A -85,B 0,C 180,E1 28389.236,E2 28389.236} C_VEL
LIN {X 0,Y 746.958,Z 852.862,A -85,B 0,C 180,E1 28386.615,E2 28386.615} C_VEL
LIN {X 0,Y 746.824,Z 907.725,A -85,B 0,C 180,E1 28385.952,E2 28385.952} C_VEL
LIN {X 0,Y 746.664,Z 934.676,A -85,B 0,C 180,E1 28385.475,E2 28385.475} C_VEL
LIN {X 0,Y 746.495,Z 961.623,A -85,B 0,C 180,E1 28384.836,E2 28384.836} C_VEL
LIN {X 0,Y 746.315,Z 984.886,A -85,B 0,C 180,E1 28384.146,E2 28384.146} C_VEL
LIN {X 0,Y 746.104,Z 1010.477,A -85,B 0,C 180,E1 28383.253,E2 28383.253} C_VEL
LIN {X 0,Y 745.82,Z 1035.181,A -85,B 0,C 180,E1 28382.225,E2 28382.225} C_VEL
LIN {X 0,Y 745.62,Z 1055.592,A -85,B 0,C 180,E1 28381.259,E2 28381.259} C_VEL
LIN {X 0,Y 745.425,Z 1075.698,A -85,B 0,C 180,E1 28380.195,E2 28380.195} C_VEL
LIN {X 0,Y 745.169,Z 1099.314,A -85,B 0,C 180,E1 28378.794,E2 28378.794} C_VEL
LIN {X 0,Y 744.942,Z 1119.882,A -85,B 0,C 180,E1 28377.408,E2 28377.408} C_VEL
LIN {X 0,Y 744.767,Z 1137.744,A -85,B 0,C 180,E1 28376.081,E2 28376.081} C_VEL
LIN {X 0,Y 744.567,Z 1157.859,A -85,B 0,C 180,E1 28374.425,E2 28374.425} C_VEL
LIN {X 0,Y 744.43,Z 1175.005,A -85,B 0,C 180,E1 28372.837,E2 28372.837} C_VEL
LIN {X 0,Y 744.307,Z 1189.643,A -85,B 0,C 180,E1 28371.346,E2 28371.346} C_VEL
LIN {X 0,Y 744.193,Z 1205.652,A -85,B 0,C 180,E1 28369.542,E2 28369.542} C_VEL
LIN {X 0,Y 744.069,Z 1220.106,A -85,B 0,C 180,E1 28367.677,E2 28367.677} C_VEL
LIN {X 0,Y 744.017,Z 1230.709,A -85,B 0,C 180,E1 28366.149,E2 28366.149} C_VEL
LIN {X 0,Y 744.006,Z 1240.608,A -85,B 0,C 180,E1 28364.552,E2 28364.552} C_VEL
LIN {X 0,Y 743.952,Z 1249.305,A -85,B 0,C 180,E1 28362.968,E2 28362.968} C_VEL
LIN {X 0,Y 743.944,Z 1257.227,A -85,B 0,C 180,E1 28361.314,E2 28361.314} C_VEL
LIN {X 0,Y 743.88,Z 1265.489,A -85,B 0,C 180,E1 28359.28,E2 28359.28} C_VEL
LIN {X 0,Y 743.917,Z 1272.577,A -85,B 0,C 180,E1 28357.023,E2 28357.023} C_VEL
LIN {X 0,Y 743.915,Z 1277.342,A -85,B 0,C 180,E1 28354.932,E2 28354.932} C_VEL
LIN {X 0,Y 743.912,Z 1280.34,A -85,B 0,C 180,E1 28352.925,E2 28352.925} C_VEL
LIN {X 0,Y 743.872,Z 1281.715,A -85,B 0,C 180,E1 28350.999,E2 28350.999} C_VEL
LIN {X 0,Y 743.863,Z 1281.826,A -85,B 0,C 180,E1 28349.382,E2 28349.382} C_VEL
LIN {X 0,Y 743.909,Z 1280.944,A -85,B 0,C 180,E1 28347.764,E2 28347.764} C_VEL
LIN {X 0,Y 743.918,Z 1278.8,A -85,B 0,C 180,E1 28345.913,E2 28345.913} C_VEL
LIN {X 0,Y 743.92,Z 1274.73,A -85,B 0,C 180,E1 28343.825,E2 28343.825} C_VEL
LIN {X 0,Y 743.91,Z 1269.322,A -85,B 0,C 180,E1 28341.885,E2 28341.885} C_VEL
LIN {X 0,Y 743.927,Z 1263.036,A -85,B 0,C 180,E1 28340.092,E2 28340.092} C_VEL
LIN {X 0,Y 743.939,Z 1256.134,A -85,B 0,C 180,E1 28338.446,E2 28338.446} C_VEL
LIN {X 0,Y 743.939,Z 1248.461,A -85,B 0,C 180,E1 28336.869,E2 28336.869} C_VEL
LIN {X 0,Y 743.997,Z 1239.651,A -85,B 0,C 180,E1 28335.284,E2 28335.284} C_VEL
LIN {X 0,Y 744.041,Z 1228.589,A -85,B 0,C 180,E1 28333.526,E2 28333.526} C_VEL
LIN {X 0,Y 744.145,Z 1214.009,A -85,B 0,C 180,E1 28331.511,E2 28331.511} C_VEL
LIN {X 0,Y 744.205,Z 1200.655,A -85,B 0,C 180,E1 28329.881,E2 28329.881} C_VEL
LIN {X 0,Y 744.328,Z 1186.984,A -85,B 0,C 180,E1 28328.373,E2 28328.373} C_VEL
LIN {X 0,Y 744.481,Z 1169.835,A -85,B 0,C 180,E1 28326.658,E2 28326.658} C_VEL
LIN {X 0,Y 744.655,Z 1150.798,A -85,B 0,C 180,E1 28324.977,E2 28324.977} C_VEL
LIN {X 0,Y 744.781,Z 1133.818,A -85,B 0,C 180,E1 28323.615,E2 28323.615} C_VEL
LIN {X 0,Y 745.052,Z 1112.486,A -85,B 0,C 180,E1 28322.07,E2 28322.07} C_VEL
LIN {X 0,Y 745.263,Z 1090.676,A -85,B 0,C 180,E1 28320.678,E2 28320.678} C_VEL
LIN {X 0,Y 745.443,Z 1071.362,A -85,B 0,C 180,E1 28319.565,E2 28319.565} C_VEL
LIN {X 0,Y 745.684,Z 1049.258,A -85,B 0,C 180,E1 28318.424,E2 28318.424} C_VEL
LIN {X 0,Y 745.969,Z 1024.263,A -85,B 0,C 180,E1 28317.303,E2 28317.303} C_VEL
LIN {X 0,Y 746.161,Z 1002.604,A -85,B 0,C 180,E1 28316.461,E2 28316.461} C_VEL
LIN {X 0,Y 746.328,Z 982.518,A -85,B 0,C 180,E1 28315.78,E2 28315.78} C_VEL
LIN {X 0,Y 746.511,Z 959.97,A -85,B 0,C 180,E1 28315.12,E2 28315.12} C_VEL
LIN {X 0,Y 746.691,Z 932.804,A -85,B 0,C 180,E1 28314.486,E2 28314.486} C_VEL
LIN {X 0,Y 746.828,Z 905.379,A -85,B 0,C 180,E1 28314.013,E2 28314.013} C_VEL
LIN {X 0,Y 747.324,Z 662.425,A -85,B 0,C 180,E1 28311.139,E2 28311.139} C_VEL
LIN {X 0,Y 747.699,Z 464.206,A -85,B 0,C 180,E1 28308.726,E2 28308.726} C_VEL
LIN {X 0,Y 747.604,Z 431.419,A -85,B 0,C 180,E1 28308.307,E2 28308.307} C_VEL
LIN {X 0,Y 746.633,Z 427.342,A -85,B 0,C 180,E1 28308.17,E2 28308.17} C_VEL
LIN {X 0,Y 746.517,Z 404.933,A -85,B 0,C 180,E1 28306.661,E2 28306.661} C_VEL
LIN {X 0,Y 745.065,Z 401.66,A -85,B 0,C 180,E1 28306.332,E2 28306.332} C_VEL
LIN {X 0,Y 743.954,Z 398.562,A -85,B 0,C 180,E1 28306.026,E2 28306.026} C_VEL
LIN {X 0,Y 743.925,Z 398.559,A -85,B 0,C 180,E1 28303.592,E2 28303.592} C_VEL
LIN {X 0,Y 743.929,Z 398.554,A -85,B 0,C 180,E1 28301.294,E2 28301.294} C_VEL
LIN {X 0,Y 743.948,Z 398.557,A -85,B 0,C 180,E1 28298.977,E2 28298.977} C_VEL
LIN {X 0,Y 744.012,Z 398.553,A -85,B 0,C 180,E1 28296.06,E2 28296.06} C_VEL
LIN {X 0,Y 743.946,Z 398.552,A -85,B 0,C 180,E1 28293.421,E2 28293.421} C_VEL
LIN {X 0,Y 743.946,Z 398.553,A -85,B 0,C 180,E1 28291.072,E2 28291.072} C_VEL
LIN {X 0,Y 743.971,Z 398.552,A -85,B 0,C 180,E1 28288.643,E2 28288.643} C_VEL
LIN {X 0,Y 743.998,Z 398.545,A -85,B 0,C 180,E1 28285.607,E2 28285.607} C_VEL
LIN {X 0,Y 743.958,Z 398.552,A -85,B 0,C 180,E1 28283.024,E2 28283.024} C_VEL
LIN {X 0,Y 743.976,Z 398.551,A -85,B 0,C 180,E1 28280.535,E2 28280.535} C_VEL
LIN {X 0,Y 744.037,Z 398.547,A -85,B 0,C 180,E1 28277.6,E2 28277.6} C_VEL
LIN {X 0,Y 743.971,Z 398.545,A -85,B 0,C 180,E1 28274.875,E2 28274.875} C_VEL
LIN {X 0,Y 743.993,Z 398.553,A -85,B 0,C 180,E1 28272.26,E2 28272.26} C_VEL
LIN {X 0,Y 744.033,Z 398.54,A -85,B 0,C 180,E1 28269.28,E2 28269.28} C_VEL
LIN {X 0,Y 743.982,Z 398.549,A -85,B 0,C 180,E1 28266.56,E2 28266.56} C_VEL
LIN {X 0,Y 744.033,Z 398.551,A -85,B 0,C 180,E1 28263.776,E2 28263.776} C_VEL
LIN {X 0,Y 744.009,Z 398.545,A -85,B 0,C 180,E1 28260.77,E2 28260.77} C_VEL
LIN {X 0,Y 744.01,Z 398.552,A -85,B 0,C 180,E1 28257.92,E2 28257.92} C_VEL
LIN {X 0,Y 744.035,Z 398.543,A -85,B 0,C 180,E1 28254.911,E2 28254.911} C_VEL
LIN {X 0,Y 744.001,Z 398.548,A -85,B 0,C 180,E1 28252.084,E2 28252.084} C_VEL
LIN {X 0,Y 744.016,Z 398.552,A -85,B 0,C 180,E1 28251.771,E2 28251.771} C_VEL
LIN {X 0,Y 743.058,Z 398.681,A -85,B 0,C 180,E1 28251.178,E2 28251.178} C_VEL
LIN {X 0,Y 736.618,Z 399.478,A -85,B 0,C 180,E1 28249.517,E2 28249.517} C_VEL
LIN {X 0,Y 736.082,Z 399.538,A -85,B 0,C 180,E1 28249.085,E2 28249.085} C_VEL
LIN {X 0,Y 736.074,Z 399.532,A -85,B 0,C 180,E1 28246.229,E2 28246.229} C_VEL
LIN {X 0,Y 736.096,Z 399.542,A -85,B 0,C 180,E1 28243.344,E2 28243.344} C_VEL
LIN {X 0,Y 736.096,Z 399.527,A -85,B 0,C 180,E1 28240.278,E2 28240.278} C_VEL
LIN {X 0,Y 736.093,Z 399.544,A -85,B 0,C 180,E1 28237.223,E2 28237.223} C_VEL
LIN {X 0,Y 736.09,Z 399.526,A -85,B 0,C 180,E1 28234.235,E2 28234.235} C_VEL
LIN {X 0,Y 736.093,Z 399.541,A -85,B 0,C 180,E1 28231.169,E2 28231.169} C_VEL
LIN {X 0,Y 736.072,Z 399.535,A -85,B 0,C 180,E1 28228.251,E2 28228.251} C_VEL
LIN {X 0,Y 736.088,Z 399.536,A -85,B 0,C 180,E1 28225.308,E2 28225.308} C_VEL
LIN {X 0,Y 736.056,Z 399.535,A -85,B 0,C 180,E1 28222.498,E2 28222.498} C_VEL
LIN {X 0,Y 736.102,Z 399.534,A -85,B 0,C 180,E1 28219.644,E2 28219.644} C_VEL
LIN {X 0,Y 736.065,Z 399.546,A -85,B 0,C 180,E1 28216.616,E2 28216.616} C_VEL
LIN {X 0,Y 736.058,Z 399.543,A -85,B 0,C 180,E1 28213.835,E2 28213.835} C_VEL
LIN {X 0,Y 736.106,Z 399.834,A -85,B 0,C 180,E1 28213.758,E2 28213.758} C_VEL
LIN {X 0,Y 737.622,Z 403.33,A -85,B 0,C 180,E1 28213.399,E2 28213.399} C_VEL
LIN {X 0,Y 740.045,Z 409.31,A -85,B 0,C 180,E1 28212.806,E2 28212.806} C_VEL
LIN {X 0,Y 740.128,Z 418.383,A -85,B 0,C 180,E1 28212.204,E2 28212.204} C_VEL
LIN {X 0,Y 741.825,Z 425.312,A -85,B 0,C 180,E1 28211.997,E2 28211.997} C_VEL
LIN {X 0,Y 741.13,Z 638.697,A -85,B 0,C 180,E1 28209.371,E2 28209.371} C_VEL
LIN {X 0,Y 740.472,Z 863.534,A -85,B 0,C 180,E1 28206.698,E2 28206.698} C_VEL
LIN {X 0,Y 740.318,Z 901.123,A -85,B 0,C 180,E1 28206.221,E2 28206.221} C_VEL
LIN {X 0,Y 740.07,Z 927.755,A -85,B 0,C 180,E1 28205.727,E2 28205.727} C_VEL
LIN {X 0,Y 739.807,Z 953.832,A -85,B 0,C 180,E1 28205.092,E2 28205.092} C_VEL
LIN {X 0,Y 739.481,Z 981.925,A -85,B 0,C 180,E1 28204.229,E2 28204.229} C_VEL
LIN {X 0,Y 739.092,Z 1006.474,A -85,B 0,C 180,E1 28203.317,E2 28203.317} C_VEL
LIN {X 0,Y 738.799,Z 1026.679,A -85,B 0,C 180,E1 28202.455,E2 28202.455} C_VEL
LIN {X 0,Y 738.501,Z 1046.392,A -85,B 0,C 180,E1 28201.509,E2 28201.509} C_VEL
LIN {X 0,Y 738.188,Z 1068.817,A -85,B 0,C 180,E1 28200.303,E2 28200.303} C_VEL
LIN {X 0,Y 737.753,Z 1092.543,A -85,B 0,C 180,E1 28198.849,E2 28198.849} C_VEL
LIN {X 0,Y 737.473,Z 1111.007,A -85,B 0,C 180,E1 28197.583,E2 28197.583} C_VEL
LIN {X 0,Y 737.207,Z 1129.886,A -85,B 0,C 180,E1 28196.156,E2 28196.156} C_VEL
LIN {X 0,Y 736.871,Z 1150.35,A -85,B 0,C 180,E1 28194.424,E2 28194.424} C_VEL
LIN {X 0,Y 736.694,Z 1166.21,A -85,B 0,C 180,E1 28192.927,E2 28192.927} C_VEL
LIN {X 0,Y 736.505,Z 1182.299,A -85,B 0,C 180,E1 28191.254,E2 28191.254} C_VEL
LIN {X 0,Y 736.305,Z 1199.146,A -85,B 0,C 180,E1 28189.27,E2 28189.27} C_VEL
LIN {X 0,Y 736.167,Z 1210.918,A -85,B 0,C 180,E1 28187.714,E2 28187.714} C_VEL
LIN {X 0,Y 736.081,Z 1221.436,A -85,B 0,C 180,E1 28186.17,E2 28186.17} C_VEL
LIN {X 0,Y 736.05,Z 1230.788,A -85,B 0,C 180,E1 28184.637,E2 28184.637} C_VEL
LIN {X 0,Y 735.98,Z 1239.873,A -85,B 0,C 180,E1 28182.955,E2 28182.955} C_VEL
LIN {X 0,Y 735.943,Z 1249.144,A -85,B 0,C 180,E1 28180.967,E2 28180.967} C_VEL
LIN {X 0,Y 735.898,Z 1257.126,A -85,B 0,C 180,E1 28178.834,E2 28178.834} C_VEL
LIN {X 0,Y 735.917,Z 1262.858,A -85,B 0,C 180,E1 28176.947,E2 28176.947} C_VEL
LIN {X 0,Y 735.912,Z 1267.544,A -85,B 0,C 180,E1 28174.834,E2 28174.834} C_VEL
LIN {X 0,Y 735.915,Z 1270.432,A -85,B 0,C 180,E1 28172.806,E2 28172.806} C_VEL
LIN {X 0,Y 735.873,Z 1271.724,A -85,B 0,C 180,E1 28170.936,E2 28170.936} C_VEL
LIN {X 0,Y 735.863,Z 1271.818,A -85,B 0,C 180,E1 28169.302,E2 28169.302} C_VEL
LIN {X 0,Y 735.904,Z 1270.919,A -85,B 0,C 180,E1 28167.666,E2 28167.666} C_VEL
LIN {X 0,Y 735.92,Z 1268.728,A -85,B 0,C 180,E1 28165.778,E2 28165.778} C_VEL
LIN {X 0,Y 735.923,Z 1264.662,A -85,B 0,C 180,E1 28163.684,E2 28163.684} C_VEL
LIN {X 0,Y 735.934,Z 1258.971,A -85,B 0,C 180,E1 28161.644,E2 28161.644} C_VEL
LIN {X 0,Y 735.945,Z 1252.923,A -85,B 0,C 180,E1 28159.909,E2 28159.909} C_VEL
LIN {X 0,Y 735.951,Z 1246.001,A -85,B 0,C 180,E1 28158.244,E2 28158.244} C_VEL
LIN {X 0,Y 735.965,Z 1238.717,A -85,B 0,C 180,E1 28156.729,E2 28156.729} C_VEL
LIN {X 0,Y 736.037,Z 1229.939,A -85,B 0,C 180,E1 28155.126,E2 28155.126} C_VEL
LIN {X 0,Y 736.109,Z 1219.955,A -85,B 0,C 180,E1 28153.51,E2 28153.51} C_VEL
LIN {X 0,Y 736.258,Z 1206.319,A -85,B 0,C 180,E1 28151.556,E2 28151.556} C_VEL
LIN {X 0,Y 736.368,Z 1191.794,A -85,B 0,C 180,E1 28149.745,E2 28149.745} C_VEL
LIN {X 0,Y 736.536,Z 1178.164,A -85,B 0,C 180,E1 28148.214,E2 28148.214} C_VEL
LIN {X 0,Y 736.718,Z 1162.9,A -85,B 0,C 180,E1 28146.656,E2 28146.656} C_VEL
LIN {X 0,Y 737.03,Z 1142.404,A -85,B 0,C 180,E1 28144.791,E2 28144.791} C_VEL
LIN {X 0,Y 737.234,Z 1125.563,A -85,B 0,C 180,E1 28143.416,E2 28143.416} C_VEL
LIN {X 0,Y 737.527,Z 1107.745,A -85,B 0,C 180,E1 28142.093,E2 28142.093} C_VEL
LIN {X 0,Y 737.939,Z 1083.68,A -85,B 0,C 180,E1 28140.497,E2 28140.497} C_VEL
LIN {X 0,Y 738.228,Z 1063.29,A -85,B 0,C 180,E1 28139.299,E2 28139.299} C_VEL
LIN {X 0,Y 738.535,Z 1043.182,A -85,B 0,C 180,E1 28138.238,E2 28138.238} C_VEL
LIN {X 0,Y 738.983,Z 1018.763,A -85,B 0,C 180,E1 28137.099,E2 28137.099} C_VEL
LIN {X 0,Y 739.315,Z 993.449,A -85,B 0,C 180,E1 28136.095,E2 28136.095} C_VEL
LIN {X 0,Y 739.578,Z 972.627,A -85,B 0,C 180,E1 28135.382,E2 28135.382} C_VEL
LIN {X 0,Y 739.853,Z 949.973,A -85,B 0,C 180,E1 28134.715,E2 28134.715} C_VEL
LIN {X 0,Y 740.127,Z 922.981,A -85,B 0,C 180,E1 28134.082,E2 28134.082} C_VEL
LIN {X 0,Y 740.334,Z 895.227,A -85,B 0,C 180,E1 28133.6,E2 28133.6} C_VEL
LIN {X 0,Y 741.07,Z 656.815,A -85,B 0,C 180,E1 28130.757,E2 28130.757} C_VEL
LIN {X 0,Y 741.705,Z 451.627,A -85,B 0,C 180,E1 28128.24,E2 28128.24} C_VEL
LIN {X 0,Y 741.656,Z 423.907,A -85,B 0,C 180,E1 28127.884,E2 28127.884} C_VEL
LIN {X 0,Y 739.978,Z 417.396,A -85,B 0,C 180,E1 28127.658,E2 28127.658} C_VEL
LIN {X 0,Y 739.948,Z 409.055,A -85,B 0,C 180,E1 28127.08,E2 28127.08} C_VEL
LIN {X 0,Y 737.097,Z 402.561,A -85,B 0,C 180,E1 28126.418,E2 28126.418} C_VEL
LIN {X 0,Y 736.044,Z 399.545,A -85,B 0,C 180,E1 28126.104,E2 28126.104} C_VEL
LIN {X 0,Y 736.032,Z 399.544,A -85,B 0,C 180,E1 28123.532,E2 28123.532} C_VEL
LIN {X 0,Y 736.1,Z 399.539,A -85,B 0,C 180,E1 28120.694,E2 28120.694} C_VEL
LIN {X 0,Y 736.037,Z 399.539,A -85,B 0,C 180,E1 28117.762,E2 28117.762} C_VEL
LIN {X 0,Y 736.027,Z 399.541,A -85,B 0,C 180,E1 28115.265,E2 28115.265} C_VEL
LIN {X 0,Y 736.089,Z 399.542,A -85,B 0,C 180,E1 28112.542,E2 28112.542} C_VEL
LIN {X 0,Y 736.04,Z 399.535,A -85,B 0,C 180,E1 28109.546,E2 28109.546} C_VEL
LIN {X 0,Y 736.021,Z 399.54,A -85,B 0,C 180,E1 28107.072,E2 28107.072} C_VEL
LIN {X 0,Y 736.053,Z 399.537,A -85,B 0,C 180,E1 28104.477,E2 28104.477} C_VEL
LIN {X 0,Y 736.055,Z 399.534,A -85,B 0,C 180,E1 28101.434,E2 28101.434} C_VEL
LIN {X 0,Y 736.018,Z 399.538,A -85,B 0,C 180,E1 28098.864,E2 28098.864} C_VEL
LIN {X 0,Y 736.028,Z 399.542,A -85,B 0,C 180,E1 28096.414,E2 28096.414} C_VEL
LIN {X 0,Y 736.101,Z 399.538,A -85,B 0,C 180,E1 28093.511,E2 28093.511} C_VEL
LIN {X 0,Y 736.02,Z 399.539,A -85,B 0,C 180,E1 28090.726,E2 28090.726} C_VEL
LIN {X 0,Y 736.016,Z 399.535,A -85,B 0,C 180,E1 28088.28,E2 28088.28} C_VEL
LIN {X 0,Y 736.072,Z 399.544,A -85,B 0,C 180,E1 28085.613,E2 28085.613} C_VEL
LIN {X 0,Y 736.032,Z 399.534,A -85,B 0,C 180,E1 28082.647,E2 28082.647} C_VEL
LIN {X 0,Y 736.011,Z 399.541,A -85,B 0,C 180,E1 28080.234,E2 28080.234} C_VEL
LIN {X 0,Y 736.013,Z 399.54,A -85,B 0,C 180,E1 28077.898,E2 28077.898} C_VEL
LIN {X 0,Y 736.069,Z 399.539,A -85,B 0,C 180,E1 28075.247,E2 28075.247} C_VEL
LIN {X 0,Y 736.027,Z 399.538,A -85,B 0,C 180,E1 28072.271,E2 28072.271} C_VEL
LIN {X 0,Y 736.006,Z 399.537,A -85,B 0,C 180,E1 28069.828,E2 28069.828} C_VEL
LIN {X 0,Y 736.011,Z 399.543,A -85,B 0,C 180,E1 28067.446,E2 28067.446} C_VEL
LIN {X 0,Y 736.098,Z 399.536,A -85,B 0,C 180,E1 28064.655,E2 28064.655} C_VEL
LIN {X 0,Y 736.014,Z 399.541,A -85,B 0,C 180,E1 28061.792,E2 28061.792} C_VEL
LIN {X 0,Y 736.001,Z 399.535,A -85,B 0,C 180,E1 28059.482,E2 28059.482} C_VEL
LIN {X 0,Y 736.001,Z 399.543,A -85,B 0,C 180,E1 28057.22,E2 28057.22} C_VEL
LIN {X 0,Y 736.028,Z 399.541,A -85,B 0,C 180,E1 28054.75,E2 28054.75} C_VEL
LIN {X 0,Y 736.026,Z 399.541,A -85,B 0,C 180,E1 28051.61,E2 28051.61} C_VEL
LIN {X 0,Y 735.999,Z 399.541,A -85,B 0,C 180,E1 28049.191,E2 28049.191} C_VEL
LIN {X 0,Y 735.995,Z 399.543,A -85,B 0,C 180,E1 28046.897,E2 28046.897} C_VEL
LIN {X 0,Y 736.003,Z 399.543,A -85,B 0,C 180,E1 28044.592,E2 28044.592} C_VEL
LIN {X 0,Y 736.092,Z 399.544,A -85,B 0,C 180,E1 28041.726,E2 28041.726} C_VEL
LIN {X 0,Y 735.998,Z 399.54,A -85,B 0,C 180,E1 28038.931,E2 28038.931} C_VEL
LIN {X 0,Y 735.992,Z 399.548,A -85,B 0,C 180,E1 28036.68,E2 28036.68} C_VEL
LIN {X 0,Y 736.002,Z 399.644,A -85,B 0,C 180,E1 28034.487,E2 28034.487} C_VEL
LIN {X 0,Y 737.273,Z 402.978,A -85,B 0,C 180,E1 28034.157,E2 28034.157} C_VEL
LIN {X 0,Y 740.17,Z 409.439,A -85,B 0,C 180,E1 28033.495,E2 28033.495} C_VEL
LIN {X 0,Y 740.194,Z 428.289,A -85,B 0,C 180,E1 28032.246,E2 28032.246} C_VEL
LIN {X 0,Y 741.772,Z 434.958,A -85,B 0,C 180,E1 28032.05,E2 28032.05} C_VEL
LIN {X 0,Y 741.181,Z 634.017,A -85,B 0,C 180,E1 28029.593,E2 28029.593} C_VEL
LIN {X 0,Y 740.518,Z 857.121,A -85,B 0,C 180,E1 28026.935,E2 28026.935} C_VEL
LIN {X 0,Y 740.322,Z 908.121,A -85,B 0,C 180,E1 28026.312,E2 28026.312} C_VEL
LIN {X 0,Y 740.086,Z 935.323,A -85,B 0,C 180,E1 28025.825,E2 28025.825} C_VEL
LIN {X 0,Y 739.83,Z 961.888,A -85,B 0,C 180,E1 28025.189,E2 28025.189} C_VEL
LIN {X 0,Y 739.549,Z 986.357,A -85,B 0,C 180,E1 28024.455,E2 28024.455} C_VEL
LIN {X 0,Y 739.196,Z 1012.079,A -85,B 0,C 180,E1 28023.539,E2 28023.539} C_VEL
LIN {X 0,Y 738.806,Z 1035.779,A -85,B 0,C 180,E1 28022.541,E2 28022.541} C_VEL
LIN {X 0,Y 738.51,Z 1055.595,A -85,B 0,C 180,E1 28021.595,E2 28021.595} C_VEL
LIN {X 0,Y 738.208,Z 1076.503,A -85,B 0,C 180,E1 28020.477,E2 28020.477} C_VEL
LIN {X 0,Y 737.787,Z 1101.306,A -85,B 0,C 180,E1 28018.976,E2 28018.976} C_VEL
LIN {X 0,Y 737.477,Z 1120.428,A -85,B 0,C 180,E1 28017.67,E2 28017.67} C_VEL
LIN {X 0,Y 737.214,Z 1138.311,A -85,B 0,C 180,E1 28016.324,E2 28016.324} C_VEL
LIN {X 0,Y 736.88,Z 1159.986,A -85,B 0,C 180,E1 28014.502,E2 28014.502} C_VEL
LIN {X 0,Y 736.693,Z 1175.86,A -85,B 0,C 180,E1 28013.006,E2 28013.006} C_VEL
LIN {X 0,Y 736.506,Z 1191.985,A -85,B 0,C 180,E1 28011.333,E2 28011.333} C_VEL
LIN {X 0,Y 736.308,Z 1208.89,A -85,B 0,C 180,E1 28009.347,E2 28009.347} C_VEL
LIN {X 0,Y 736.17,Z 1220.69,A -85,B 0,C 180,E1 28007.791,E2 28007.791} C_VEL
LIN {X 0,Y 736.087,Z 1231.233,A -85,B 0,C 180,E1 28006.247,E2 28006.247} C_VEL
LIN {X 0,Y 736.049,Z 1241.075,A -85,B 0,C 180,E1 28004.633,E2 28004.633} C_VEL
LIN {X 0,Y 735.992,Z 1250.538,A -85,B 0,C 180,E1 28002.871,E2 28002.871} C_VEL
LIN {X 0,Y 735.933,Z 1260.606,A -85,B 0,C 180,E1 28000.645,E2 28000.645} C_VEL
LIN {X 0,Y 735.902,Z 1267.288,A -85,B 0,C 180,E1 27998.829,E2 27998.829} C_VEL
LIN {X 0,Y 735.916,Z 1272.985,A -85,B 0,C 180,E1 27996.943,E2 27996.943} C_VEL
LIN {X 0,Y 735.912,Z 1277.638,A -85,B 0,C 180,E1 27994.83,E2 27994.83} C_VEL
LIN {X 0,Y 735.914,Z 1280.408,A -85,B 0,C 180,E1 27992.879,E2 27992.879} C_VEL
LIN {X 0,Y 735.873,Z 1281.715,A -85,B 0,C 180,E1 27991.01,E2 27991.01} C_VEL
LIN {X 0,Y 735.863,Z 1281.826,A -85,B 0,C 180,E1 27989.375,E2 27989.375} C_VEL
LIN {X 0,Y 735.908,Z 1280.944,A -85,B 0,C 180,E1 27987.74,E2 27987.74} C_VEL
LIN {X 0,Y 735.918,Z 1278.8,A -85,B 0,C 180,E1 27985.868,E2 27985.868} C_VEL
LIN {X 0,Y 735.923,Z 1274.73,A -85,B 0,C 180,E1 27983.758,E2 27983.758} C_VEL
LIN {X 0,Y 735.932,Z 1269.066,A -85,B 0,C 180,E1 27981.718,E2 27981.718} C_VEL
LIN {X 0,Y 735.945,Z 1263.037,A -85,B 0,C 180,E1 27979.983,E2 27979.983} C_VEL
LIN {X 0,Y 735.951,Z 1256.135,A -85,B 0,C 180,E1 27978.319,E2 27978.319} C_VEL
LIN {X 0,Y 735.966,Z 1248.873,A -85,B 0,C 180,E1 27976.805,E2 27976.805} C_VEL
LIN {X 0,Y 736.041,Z 1240.118,A -85,B 0,C 180,E1 27975.202,E2 27975.202} C_VEL
LIN {X 0,Y 736.105,Z 1229.836,A -85,B 0,C 180,E1 27973.537,E2 27973.537} C_VEL
LIN {X 0,Y 736.259,Z 1215.934,A -85,B 0,C 180,E1 27971.551,E2 27971.551} C_VEL
LIN {X 0,Y 736.374,Z 1201.367,A -85,B 0,C 180,E1 27969.74,E2 27969.74} C_VEL
LIN {X 0,Y 736.538,Z 1187.742,A -85,B 0,C 180,E1 27968.213,E2 27968.213} C_VEL
LIN {X 0,Y 736.753,Z 1171.418,A -85,B 0,C 180,E1 27966.555,E2 27966.555} C_VEL
LIN {X 0,Y 737.035,Z 1151.813,A -85,B 0,C 180,E1 27964.786,E2 27964.786} C_VEL
LIN {X 0,Y 737.239,Z 1134.925,A -85,B 0,C 180,E1 27963.411,E2 27963.411} C_VEL
LIN {X 0,Y 737.583,Z 1115.578,A -85,B 0,C 180,E1 27961.982,E2 27961.982} C_VEL
LIN {X 0,Y 737.955,Z 1092.084,A -85,B 0,C 180,E1 27960.445,E2 27960.445} C_VEL
LIN {X 0,Y 738.234,Z 1072.395,A -85,B 0,C 180,E1 27959.294,E2 27959.294} C_VEL
LIN {X 0,Y 738.554,Z 1051.931,A -85,B 0,C 180,E1 27958.22,E2 27958.22} C_VEL
LIN {X 0,Y 739.02,Z 1025.791,A -85,B 0,C 180,E1 27957.02,E2 27957.02} C_VEL
LIN {X 0,Y 739.317,Z 1003.349,A -85,B 0,C 180,E1 27956.136,E2 27956.136} C_VEL
LIN {X 0,Y 739.58,Z 982.462,A -85,B 0,C 180,E1 27955.422,E2 27955.422} C_VEL
LIN {X 0,Y 739.855,Z 959.845,A -85,B 0,C 180,E1 27954.757,E2 27954.757} C_VEL
LIN {X 0,Y 740.13,Z 932.837,A -85,B 0,C 180,E1 27954.124,E2 27954.124} C_VEL
LIN {X 0,Y 740.335,Z 905.181,A -85,B 0,C 180,E1 27953.645,E2 27953.645} C_VEL
LIN {X 0,Y 741.074,Z 665.853,A -85,B 0,C 180,E1 27950.791,E2 27950.791} C_VEL
LIN {X 0,Y 741.663,Z 467.507,A -85,B 0,C 180,E1 27948.357,E2 27948.357} C_VEL
LIN {X 0,Y 741.605,Z 433.593,A -85,B 0,C 180,E1 27947.921,E2 27947.921} C_VEL
LIN {X 0,Y 740.051,Z 427.342,A -85,B 0,C 180,E1 27947.712,E2 27947.712} C_VEL
